LIN {X 0,Y 176.347,Z 623.439,A -85,B 0,C 180,E1 -22419.173,E2 -22419.173} C_VEL
LIN {X 0,Y 177.506,Z 621.11,A -85,B 0,C 180,E1 -22423.742,E2 -22423.742} C_VEL
LIN {X 0,Y 179.733,Z 617.398,A -85,B 0,C 180,E1 -22428.229,E2 -22428.229} C_VEL
LIN {X 0,Y 182.863,Z 612.047,A -85,B 0,C 180,E1 -22432.722,E2 -22432.722} C_VEL
LIN {X 0,Y 186.944,Z 605.294,A -85,B 0,C 180,E1 -22436.815,E2 -22436.815} C_VEL
LIN {X 0,Y 191.406,Z 597.669,A -85,B 0,C 180,E1 -22440.322,E2 -22440.322} C_VEL
LIN {X 0,Y 195.831,Z 589.742,A -85,B 0,C 180,E1 -22443.18,E2 -22443.18} C_VEL
LIN {X 0,Y 200.702,Z 580.202,A -85,B 0,C 180,E1 -22445.911,E2 -22445.911} C_VEL
LIN {X 0,Y 205.489,Z 569.651,A -85,B 0,C 180,E1 -22448.308,E2 -22448.308} C_VEL
LIN {X 0,Y 210.252,Z 558.007,A -85,B 0,C 180,E1 -22450.363,E2 -22450.363} C_VEL
LIN {X 0,Y 214.231,Z 546.657,A -85,B 0,C 180,E1 -22451.943,E2 -22451.943} C_VEL
LIN {X 0,Y 217.948,Z 534.375,A -85,B 0,C 180,E1 -22453.252,E2 -22453.252} C_VEL
LIN {X 0,Y 221.215,Z 520.802,A -85,B 0,C 180,E1 -22454.34,E2 -22454.34} C_VEL
LIN {X 0,Y 223.705,Z 506.759,A -85,B 0,C 180,E1 -22455.138,E2 -22455.138} C_VEL
LIN {X 0,Y 225.13,Z 493.571,A -85,B 0,C 180,E1 -22455.648,E2 -22455.648} C_VEL
LIN {X 0,Y 228.62,Z 440.792,A -85,B 0,C 180,E1 -22457.146,E2 -22457.146} C_VEL
LIN {X 0,Y 223.879,Z 429.35,A -85,B 0,C 180,E1 -22459.176,E2 -22459.176} C_VEL
LIN {X 0,Y 218.405,Z 417.952,A -85,B 0,C 180,E1 -22461.66,E2 -22461.66} C_VEL
LIN {X 0,Y 213.133,Z 408.172,A -85,B 0,C 180,E1 -22464.263,E2 -22464.263} C_VEL
LIN {X 0,Y 208.258,Z 399.763,A -85,B 0,C 180,E1 -22466.934,E2 -22466.934} C_VEL
LIN {X 0,Y 204.902,Z 394.49,A -85,B 0,C 180,E1 -22468.95,E2 -22468.95} C_VEL
LIN {X 0,Y 201.919,Z 389.944,A -85,B 0,C 180,E1 -22470.91,E2 -22470.91} C_VEL
LIN {X 0,Y 198.244,Z 384.689,A -85,B 0,C 180,E1 -22473.59,E2 -22473.59} C_VEL
LIN {X 0,Y 195.498,Z 381.922,A -85,B 0,C 180,E1 -22475.76,E2 -22475.76} C_VEL
LIN {X 0,Y 194.093,Z 379.464,A -85,B 0,C 180,E1 -22477.093,E2 -22477.093} C_VEL
LIN {X 0,Y 191.265,Z 377.162,A -85,B 0,C 180,E1 -22479.815,E2 -22479.815} C_VEL
LIN {X 0,Y 189.615,Z 374.053,A -85,B 0,C 180,E1 -22481.903,E2 -22481.903} C_VEL
LIN {X 0,Y 186.176,Z 371.524,A -85,B 0,C 180,E1 -22486.91,E2 -22486.91} C_VEL
LIN {X 0,Y 185.017,Z 368.902,A -85,B 0,C 180,E1 -22489.847,E2 -22489.847} C_VEL
LIN {X 0,Y 184.851,Z 367.99,A -85,B 0,C 180,E1 -22490.546,E2 -22490.546} C_VEL
LIN {X 0,Y 183.865,Z 367.537,A -85,B 0,C 180,E1 -22500.001,E2 -22500.001} C_VEL
LIN {X 0,Y 184.86,Z 368.103,A -85,B 0,C 180,E1 -22503.952,E2 -22503.952} C_VEL
LIN {X 0,Y 186.113,Z 371.068,A -85,B 0,C 180,E1 -22507.323,E2 -22507.323} C_VEL
LIN {X 0,Y 188.809,Z 373.526,A -85,B 0,C 180,E1 -22511.542,E2 -22511.542} C_VEL
LIN {X 0,Y 189.74,Z 374.056,A -85,B 0,C 180,E1 -22512.671,E2 -22512.671} C_VEL
LIN {X 0,Y 191.233,Z 376.977,A -85,B 0,C 180,E1 -22514.568,E2 -22514.568} C_VEL
LIN {X 0,Y 194.282,Z 379.772,A -85,B 0,C 180,E1 -22517.526,E2 -22517.526} C_VEL
LIN {X 0,Y 196.429,Z 383.09,A -85,B 0,C 180,E1 -22519.463,E2 -22519.463} C_VEL
LIN {X 0,Y 198.609,Z 385.225,A -85,B 0,C 180,E1 -22521.131,E2 -22521.131} C_VEL
LIN {X 0,Y 201.298,Z 388.85,A -85,B 0,C 180,E1 -22523.083,E2 -22523.083} C_VEL
LIN {X 0,Y 202.611,Z 390.385,A -85,B 0,C 180,E1 -22523.951,E2 -22523.951} C_VEL
LIN {X 0,Y 206.418,Z 395.562,A -85,B 0,C 180,E1 -22526.329,E2 -22526.329} C_VEL
LIN {X 0,Y 210.161,Z 400.809,A -85,B 0,C 180,E1 -22528.441,E2 -22528.441} C_VEL
LIN {X 0,Y 214.285,Z 406.702,A -85,B 0,C 180,E1 -22530.555,E2 -22530.555} C_VEL
LIN {X 0,Y 221.11,Z 417.678,A -85,B 0,C 180,E1 -22533.724,E2 -22533.724} C_VEL
LIN {X 0,Y 224.783,Z 424.595,A -85,B 0,C 180,E1 -22535.312,E2 -22535.312} C_VEL
LIN {X 0,Y 229.084,Z 433.995,A -85,B 0,C 180,E1 -22537.104,E2 -22537.104} C_VEL
LIN {X 0,Y 225.117,Z 490.442,A -85,B 0,C 180,E1 -22538.697,E2 -22538.697} C_VEL
LIN {X 0,Y 223.295,Z 504.424,A -85,B 0,C 180,E1 -22539.378,E2 -22539.378} C_VEL
LIN {X 0,Y 220.715,Z 518.004,A -85,B 0,C 180,E1 -22540.342,E2 -22540.342} C_VEL
LIN {X 0,Y 217.324,Z 531.263,A -85,B 0,C 180,E1 -22541.599,E2 -22541.599} C_VEL
LIN {X 0,Y 213.305,Z 544.035,A -85,B 0,C 180,E1 -22543.201,E2 -22543.201} C_VEL
LIN {X 0,Y 208.902,Z 555.625,A -85,B 0,C 180,E1 -22545.051,E2 -22545.051} C_VEL
LIN {X 0,Y 204.242,Z 566.232,A -85,B 0,C 180,E1 -22547.189,E2 -22547.189} C_VEL
LIN {X 0,Y 199.25,Z 576.745,A -85,B 0,C 180,E1 -22549.932,E2 -22549.932} C_VEL
LIN {X 0,Y 194.962,Z 584.9,A -85,B 0,C 180,E1 -22552.627,E2 -22552.627} C_VEL
LIN {X 0,Y 190.644,Z 592.537,A -85,B 0,C 180,E1 -22555.794,E2 -22555.794} C_VEL
LIN {X 0,Y 186.448,Z 599.361,A -85,B 0,C 180,E1 -22559.412,E2 -22559.412} C_VEL
LIN {X 0,Y 182.571,Z 605.398,A -85,B 0,C 180,E1 -22563.725,E2 -22563.725} C_VEL
LIN {X 0,Y 180.255,Z 608.851,A -85,B 0,C 180,E1 -22567.053,E2 -22567.053} C_VEL
LIN {X 0,Y 178.042,Z 612.15,A -85,B 0,C 180,E1 -22571.592,E2 -22571.592} C_VEL
LIN {X 0,Y 176.557,Z 614.028,A -85,B 0,C 180,E1 -22576.183,E2 -22576.183} C_VEL
LIN {X 0,Y 175.955,Z 614.552,A -85,B 0,C 180,E1 -22580.807,E2 -22580.807} C_VEL
LIN {X 0,Y 176.019,Z 613.752,A -85,B 0,C 180,E1 -22585.42,E2 -22585.42} C_VEL
LIN {X 0,Y 176.277,Z 611.638,A -85,B 0,C 180,E1 -22590,E2 -22590} C_VEL
LIN {X 0,Y 177.061,Z 608.156,A -85,B 0,C 180,E1 -22594.553,E2 -22594.553} C_VEL
LIN {X 0,Y 178.635,Z 603.197,A -85,B 0,C 180,E1 -22599.054,E2 -22599.054} C_VEL
LIN {X 0,Y 180.415,Z 598.399,A -85,B 0,C 180,E1 -22602.371,E2 -22602.371} C_VEL
LIN {X 0,Y 182.925,Z 591.954,A -85,B 0,C 180,E1 -22605.931,E2 -22605.931} C_VEL
LIN {X 0,Y 185.824,Z 584.276,A -85,B 0,C 180,E1 -22609.325,E2 -22609.325} C_VEL
LIN {X 0,Y 189.093,Z 575.604,A -85,B 0,C 180,E1 -22612.392,E2 -22612.392} C_VEL
LIN {X 0,Y 192.844,Z 565.1,A -85,B 0,C 180,E1 -22615.354,E2 -22615.354} C_VEL
LIN {X 0,Y 196.711,Z 553.334,A -85,B 0,C 180,E1 -22617.964,E2 -22617.964} C_VEL
LIN {X 0,Y 200.089,Z 541.52,A -85,B 0,C 180,E1 -22620.034,E2 -22620.034} C_VEL
LIN {X 0,Y 202.809,Z 530.234,A -85,B 0,C 180,E1 -22621.609,E2 -22621.609} C_VEL
LIN {X 0,Y 205.621,Z 517.023,A -85,B 0,C 180,E1 -22623.005,E2 -22623.005} C_VEL
LIN {X 0,Y 207.715,Z 503.456,A -85,B 0,C 180,E1 -22624.082,E2 -22624.082} C_VEL
LIN {X 0,Y 209.146,Z 489.592,A -85,B 0,C 180,E1 -22624.837,E2 -22624.837} C_VEL
LIN {X 0,Y 213.093,Z 419.656,A -85,B 0,C 180,E1 -22627.034,E2 -22627.034} C_VEL
LIN {X 0,Y 208.609,Z 408.771,A -85,B 0,C 180,E1 -22628.586,E2 -22628.586} C_VEL
LIN {X 0,Y 200.689,Z 394.452,A -85,B 0,C 180,E1 -22631.361,E2 -22631.361} C_VEL
LIN {X 0,Y 193.602,Z 383.533,A -85,B 0,C 180,E1 -22634.066,E2 -22634.066} C_VEL
LIN {X 0,Y 188.109,Z 375.762,A -85,B 0,C 180,E1 -22636.369,E2 -22636.369} C_VEL
LIN {X 0,Y 185.242,Z 371.796,A -85,B 0,C 180,E1 -22637.667,E2 -22637.667} C_VEL
LIN {X 0,Y 182.829,Z 368.831,A -85,B 0,C 180,E1 -22638.797,E2 -22638.797} C_VEL
LIN {X 0,Y 181.921,Z 367.135,A -85,B 0,C 180,E1 -22639.275,E2 -22639.275} C_VEL
LIN {X 0,Y 179.566,Z 364.991,A -85,B 0,C 180,E1 -22640.413,E2 -22640.413} C_VEL
LIN {X 0,Y 178.526,Z 362.549,A -85,B 0,C 180,E1 -22641.036,E2 -22641.036} C_VEL
LIN {X 0,Y 178.411,Z 361.88,A -85,B 0,C 180,E1 -22641.24,E2 -22641.24} C_VEL
LIN {X 0,Y 178.483,Z 361.865,A -85,B 0,C 180,E1 -22646.545,E2 -22646.545} C_VEL
LIN {X 0,Y 178.519,Z 361.868,A -85,B 0,C 180,E1 -22650.006,E2 -22650.006} C_VEL
LIN {X 0,Y 178.517,Z 361.866,A -85,B 0,C 180,E1 -22654.885,E2 -22654.885} C_VEL
LIN {X 0,Y 178.603,Z 361.846,A -85,B 0,C 180,E1 -22661.65,E2 -22661.65} C_VEL
LIN {X 0,Y 178.633,Z 361.829,A -85,B 0,C 180,E1 -22666.345,E2 -22666.345} C_VEL
LIN {X 0,Y 178.901,Z 361.824,A -85,B 0,C 180,E1 -22670.958,E2 -22670.958} C_VEL
LIN {X 0,Y 179.119,Z 361.78,A -85,B 0,C 180,E1 -22677.751,E2 -22677.751} C_VEL
LIN {X 0,Y 179.332,Z 361.773,A -85,B 0,C 180,E1 -22679.999,E2 -22679.999} C_VEL
LIN {X 0,Y 178.884,Z 361.827,A -85,B 0,C 180,E1 -22686.768,E2 -22686.768} C_VEL
LIN {X 0,Y 178.827,Z 361.819,A -85,B 0,C 180,E1 -22690.74,E2 -22690.74} C_VEL
LIN {X 0,Y 178.585,Z 361.846,A -85,B 0,C 180,E1 -22695.99,E2 -22695.99} C_VEL
LIN {X 0,Y 178.552,Z 361.864,A -85,B 0,C 180,E1 -22699.154,E2 -22699.154} C_VEL
LIN {X 0,Y 178.51,Z 361.862,A -85,B 0,C 180,E1 -22705.111,E2 -22705.111} C_VEL
LIN {X 0,Y 178.455,Z 361.87,A -85,B 0,C 180,E1 -22710.795,E2 -22710.795} C_VEL
LIN {X 0,Y 178.47,Z 361.887,A -85,B 0,C 180,E1 -22712.531,E2 -22712.531} C_VEL
LIN {X 0,Y 179.25,Z 364.296,A -85,B 0,C 180,E1 -22713.04,E2 -22713.04} C_VEL
LIN {X 0,Y 181.077,Z 366.543,A -85,B 0,C 180,E1 -22713.972,E2 -22713.972} C_VEL
LIN {X 0,Y 182.337,Z 367.607,A -85,B 0,C 180,E1 -22714.562,E2 -22714.562} C_VEL
LIN {X 0,Y 184.25,Z 370.718,A -85,B 0,C 180,E1 -22715.52,E2 -22715.52} C_VEL
LIN {X 0,Y 185.968,Z 372.684,A -85,B 0,C 180,E1 -22716.297,E2 -22716.297} C_VEL
LIN {X 0,Y 188.777,Z 376.476,A -85,B 0,C 180,E1 -22717.546,E2 -22717.546} C_VEL
LIN {X 0,Y 194.692,Z 386.533,A -85,B 0,C 180,E1 -22720.08,E2 -22720.08} C_VEL
LIN {X 0,Y 201.001,Z 398.408,A -85,B 0,C 180,E1 -22722.559,E2 -22722.559} C_VEL
LIN {X 0,Y 206.826,Z 411.246,A -85,B 0,C 180,E1 -22724.717,E2 -22724.717} C_VEL
LIN {X 0,Y 212.704,Z 426.479,A -85,B 0,C 180,E1 -22726.81,E2 -22726.81} C_VEL
LIN {X 0,Y 212.485,Z 434.308,A -85,B 0,C 180,E1 -22727.099,E2 -22727.099} C_VEL
LIN {X 0,Y 210.836,Z 461.914,A -85,B 0,C 180,E1 -22727.922,E2 -22727.922} C_VEL
LIN {X 0,Y 209.983,Z 467.763,A -85,B 0,C 180,E1 -22727.981,E2 -22727.981} C_VEL
LIN {X 0,Y 204.53,Z 486.79,A -85,B 0,C 180,E1 -22727.57,E2 -22727.57} C_VEL
LIN {X 0,Y 203.628,Z 492.629,A -85,B 0,C 180,E1 -22727.646,E2 -22727.646} C_VEL
LIN {X 0,Y 202.346,Z 506.62,A -85,B 0,C 180,E1 -22728.254,E2 -22728.254} C_VEL
LIN {X 0,Y 200.244,Z 520.531,A -85,B 0,C 180,E1 -22729.181,E2 -22729.181} C_VEL
LIN {X 0,Y 197.387,Z 534.321,A -85,B 0,C 180,E1 -22730.474,E2 -22730.474} C_VEL
LIN {X 0,Y 194.258,Z 546.758,A -85,B 0,C 180,E1 -22732.047,E2 -22732.047} C_VEL
LIN {X 0,Y 190.491,Z 559.651,A -85,B 0,C 180,E1 -22734.176,E2 -22734.176} C_VEL
LIN {X 0,Y 186.997,Z 569.993,A -85,B 0,C 180,E1 -22736.335,E2 -22736.335} C_VEL
LIN {X 0,Y 183.467,Z 579.723,A -85,B 0,C 180,E1 -22738.86,E2 -22738.86} C_VEL
LIN {X 0,Y 179.689,Z 589.461,A -85,B 0,C 180,E1 -22742.009,E2 -22742.009} C_VEL
LIN {X 0,Y 176.498,Z 597.532,A -85,B 0,C 180,E1 -22745.286,E2 -22745.286} C_VEL
LIN {X 0,Y 173.566,Z 605.272,A -85,B 0,C 180,E1 -22749.25,E2 -22749.25} C_VEL
LIN {X 0,Y 171.381,Z 611.465,A -85,B 0,C 180,E1 -22753.319,E2 -22753.319} C_VEL
LIN {X 0,Y 170.039,Z 615.675,A -85,B 0,C 180,E1 -22756.861,E2 -22756.861} C_VEL
LIN {X 0,Y 169.291,Z 619.025,A -85,B 0,C 180,E1 -22760.442,E2 -22760.442} C_VEL
LIN {X 0,Y 168.872,Z 622.15,A -85,B 0,C 180,E1 -22765.226,E2 -22765.226} C_VEL
LIN {X 0,Y 168.885,Z 623.187,A -85,B 0,C 180,E1 -22767.615,E2 -22767.615} C_VEL
LIN {X 0,Y 168.999,Z 623.881,A -85,B 0,C 180,E1 -22770,E2 -22770} C_VEL
LIN {X 0,Y 168.857,Z 624.241,A -85,B 0,C 180,E1 -22774.775,E2 -22774.775} C_VEL
LIN {X 0,Y 169.315,Z 623.275,A -85,B 0,C 180,E1 -22779.557,E2 -22779.557} C_VEL
LIN {X 0,Y 170.568,Z 620.977,A -85,B 0,C 180,E1 -22784.313,E2 -22784.313} C_VEL
LIN {X 0,Y 172.941,Z 617.296,A -85,B 0,C 180,E1 -22788.971,E2 -22788.971} C_VEL
LIN {X 0,Y 176.187,Z 612.126,A -85,B 0,C 180,E1 -22793.508,E2 -22793.508} C_VEL
LIN {X 0,Y 179.414,Z 607.14,A -85,B 0,C 180,E1 -22796.774,E2 -22796.774} C_VEL
LIN {X 0,Y 183.861,Z 600.02,A -85,B 0,C 180,E1 -22800.428,E2 -22800.428} C_VEL
LIN {X 0,Y 188.274,Z 592.588,A -85,B 0,C 180,E1 -22803.407,E2 -22803.407} C_VEL
LIN {X 0,Y 193.292,Z 583.68,A -85,B 0,C 180,E1 -22806.216,E2 -22806.216} C_VEL
LIN {X 0,Y 198.071,Z 573.961,A -85,B 0,C 180,E1 -22808.684,E2 -22808.684} C_VEL
LIN {X 0,Y 202.892,Z 563.197,A -85,B 0,C 180,E1 -22810.828,E2 -22810.828} C_VEL
LIN {X 0,Y 207.421,Z 551.539,A -85,B 0,C 180,E1 -22812.659,E2 -22812.659} C_VEL
LIN {X 0,Y 211.743,Z 538.704,A -85,B 0,C 180,E1 -22814.186,E2 -22814.186} C_VEL
LIN {X 0,Y 215.364,Z 525.362,A -85,B 0,C 180,E1 -22815.381,E2 -22815.381} C_VEL
LIN {X 0,Y 218.181,Z 511.58,A -85,B 0,C 180,E1 -22816.28,E2 -22816.28} C_VEL
LIN {X 0,Y 220.114,Z 497.18,A -85,B 0,C 180,E1 -22816.916,E2 -22816.916} C_VEL
LIN {X 0,Y 223.975,Z 443.363,A -85,B 0,C 180,E1 -22818.439,E2 -22818.439} C_VEL
LIN {X 0,Y 219.593,Z 432.728,A -85,B 0,C 180,E1 -22820.437,E2 -22820.437} C_VEL
LIN {X 0,Y 214.834,Z 422.604,A -85,B 0,C 180,E1 -22822.734,E2 -22822.734} C_VEL
LIN {X 0,Y 209.923,Z 413.205,A -85,B 0,C 180,E1 -22825.31,E2 -22825.31} C_VEL
LIN {X 0,Y 204.972,Z 404.476,A -85,B 0,C 180,E1 -22828.202,E2 -22828.202} C_VEL
LIN {X 0,Y 202.27,Z 400.161,A -85,B 0,C 180,E1 -22829.928,E2 -22829.928} C_VEL
LIN {X 0,Y 199.369,Z 395.626,A -85,B 0,C 180,E1 -22831.951,E2 -22831.951} C_VEL
LIN {X 0,Y 196.225,Z 391.115,A -85,B 0,C 180,E1 -22834.369,E2 -22834.369} C_VEL
LIN {X 0,Y 193.505,Z 388.049,A -85,B 0,C 180,E1 -22836.665,E2 -22836.665} C_VEL
LIN {X 0,Y 192.296,Z 386.084,A -85,B 0,C 180,E1 -22837.859,E2 -22837.859} C_VEL
LIN {X 0,Y 189.57,Z 383.514,A -85,B 0,C 180,E1 -22840.676,E2 -22840.676} C_VEL
LIN {X 0,Y 188.133,Z 380.752,A -85,B 0,C 180,E1 -22842.612,E2 -22842.612} C_VEL
LIN {X 0,Y 185.178,Z 378.541,A -85,B 0,C 180,E1 -22847.117,E2 -22847.117} C_VEL
LIN {X 0,Y 183.971,Z 375.813,A -85,B 0,C 180,E1 -22850.314,E2 -22850.314} C_VEL
LIN {X 0,Y 183.753,Z 374.963,A -85,B 0,C 180,E1 -22851.201,E2 -22851.201} C_VEL
LIN {X 0,Y 182.999,Z 374.568,A -85,B 0,C 180,E1 -22860.001,E2 -22860.001} C_VEL
LIN {X 0,Y 183.852,Z 375.08,A -85,B 0,C 180,E1 -22863.562,E2 -22863.562} C_VEL
LIN {X 0,Y 185.105,Z 378.074,A -85,B 0,C 180,E1 -22867.089,E2 -22867.089} C_VEL
LIN {X 0,Y 187.956,Z 380.602,A -85,B 0,C 180,E1 -22871.595,E2 -22871.595} C_VEL
LIN {X 0,Y 188.5,Z 381.338,A -85,B 0,C 180,E1 -22872.329,E2 -22872.329} C_VEL
LIN {X 0,Y 190.352,Z 384.369,A -85,B 0,C 180,E1 -22874.637,E2 -22874.637} C_VEL
LIN {X 0,Y 192.699,Z 386.55,A -85,B 0,C 180,E1 -22876.965,E2 -22876.965} C_VEL
LIN {X 0,Y 194.824,Z 389.778,A -85,B 0,C 180,E1 -22878.946,E2 -22878.946} C_VEL
LIN {X 0,Y 196.77,Z 391.782,A -85,B 0,C 180,E1 -22880.5,E2 -22880.5} C_VEL
LIN {X 0,Y 199.598,Z 395.55,A -85,B 0,C 180,E1 -22882.618,E2 -22882.618} C_VEL
LIN {X 0,Y 204.059,Z 401.66,A -85,B 0,C 180,E1 -22885.569,E2 -22885.569} C_VEL
LIN {X 0,Y 209.178,Z 409.019,A -85,B 0,C 180,E1 -22888.531,E2 -22888.531} C_VEL
LIN {X 0,Y 214.446,Z 417.321,A -85,B 0,C 180,E1 -22891.245,E2 -22891.245} C_VEL
LIN {X 0,Y 219.675,Z 426.375,A -85,B 0,C 180,E1 -22893.689,E2 -22893.689} C_VEL
LIN {X 0,Y 224.384,Z 436.682,A -85,B 0,C 180,E1 -22895.793,E2 -22895.793} C_VEL
LIN {X 0,Y 220.468,Z 490.541,A -85,B 0,C 180,E1 -22897.325,E2 -22897.325} C_VEL
LIN {X 0,Y 218.601,Z 504.443,A -85,B 0,C 180,E1 -22898.001,E2 -22898.001} C_VEL
LIN {X 0,Y 215.865,Z 518.316,A -85,B 0,C 180,E1 -22898.987,E2 -22898.987} C_VEL
LIN {X 0,Y 212.103,Z 532.442,A -85,B 0,C 180,E1 -22900.352,E2 -22900.352} C_VEL
LIN {X 0,Y 207.937,Z 545.022,A -85,B 0,C 180,E1 -22901.965,E2 -22901.965} C_VEL
LIN {X 0,Y 203.366,Z 556.527,A -85,B 0,C 180,E1 -22903.847,E2 -22903.847} C_VEL
LIN {X 0,Y 198.103,Z 567.943,A -85,B 0,C 180,E1 -22906.23,E2 -22906.23} C_VEL
LIN {X 0,Y 192.935,Z 578.139,A -85,B 0,C 180,E1 -22909.03,E2 -22909.03} C_VEL
LIN {X 0,Y 188.108,Z 586.801,A -85,B 0,C 180,E1 -22912.068,E2 -22912.068} C_VEL
LIN {X 0,Y 183.371,Z 594.596,A -85,B 0,C 180,E1 -22915.577,E2 -22915.577} C_VEL
LIN {X 0,Y 179.128,Z 601.026,A -85,B 0,C 180,E1 -22919.334,E2 -22919.334} C_VEL
LIN {X 0,Y 175.196,Z 606.7,A -85,B 0,C 180,E1 -22923.816,E2 -22923.816} C_VEL
LIN {X 0,Y 172.28,Z 610.785,A -85,B 0,C 180,E1 -22928.461,E2 -22928.461} C_VEL
LIN {X 0,Y 170.278,Z 613.41,A -85,B 0,C 180,E1 -22933.207,E2 -22933.207} C_VEL
LIN {X 0,Y 169.121,Z 614.65,A -85,B 0,C 180,E1 -22938.008,E2 -22938.008} C_VEL
LIN {X 0,Y 168.831,Z 614.547,A -85,B 0,C 180,E1 -22942.826,E2 -22942.826} C_VEL
LIN {X 0,Y 168.983,Z 613.555,A -85,B 0,C 180,E1 -22946.543,E2 -22946.543} C_VEL
LIN {X 0,Y 169.177,Z 611.922,A -85,B 0,C 180,E1 -22950,E2 -22950} C_VEL
LIN {X 0,Y 170.002,Z 608.478,A -85,B 0,C 180,E1 -22954.743,E2 -22954.743} C_VEL
LIN {X 0,Y 171.648,Z 603.56,A -85,B 0,C 180,E1 -22959.426,E2 -22959.426} C_VEL
LIN {X 0,Y 173.514,Z 598.806,A -85,B 0,C 180,E1 -22962.871,E2 -22962.871} C_VEL
LIN {X 0,Y 176.126,Z 592.409,A -85,B 0,C 180,E1 -22966.563,E2 -22966.563} C_VEL
LIN {X 0,Y 179.164,Z 584.785,A -85,B 0,C 180,E1 -22970.073,E2 -22970.073} C_VEL
LIN {X 0,Y 182.581,Z 576.175,A -85,B 0,C 180,E1 -22973.237,E2 -22973.237} C_VEL
LIN {X 0,Y 186.482,Z 565.745,A -85,B 0,C 180,E1 -22976.283,E2 -22976.283} C_VEL
LIN {X 0,Y 190.512,Z 554.068,A -85,B 0,C 180,E1 -22978.958,E2 -22978.958} C_VEL
LIN {X 0,Y 194.008,Z 542.371,A -85,B 0,C 180,E1 -22981.077,E2 -22981.077} C_VEL
LIN {X 0,Y 196.833,Z 531.239,A -85,B 0,C 180,E1 -22982.686,E2 -22982.686} C_VEL
LIN {X 0,Y 199.719,Z 518.257,A -85,B 0,C 180,E1 -22984.112,E2 -22984.112} C_VEL
LIN {X 0,Y 202.031,Z 504.288,A -85,B 0,C 180,E1 -22985.256,E2 -22985.256} C_VEL
LIN {X 0,Y 203.634,Z 489.716,A -85,B 0,C 180,E1 -22986.068,E2 -22986.068} C_VEL
LIN {X 0,Y 207.648,Z 421.746,A -85,B 0,C 180,E1 -22988.234,E2 -22988.234} C_VEL
LIN {X 0,Y 203.963,Z 412.813,A -85,B 0,C 180,E1 -22989.582,E2 -22989.582} C_VEL
LIN {X 0,Y 196.447,Z 399.021,A -85,B 0,C 180,E1 -22992.367,E2 -22992.367} C_VEL
LIN {X 0,Y 189.899,Z 388.695,A -85,B 0,C 180,E1 -22995.008,E2 -22995.008} C_VEL
LIN {X 0,Y 184.401,Z 380.876,A -85,B 0,C 180,E1 -22997.439,E2 -22997.439} C_VEL
LIN {X 0,Y 181.917,Z 377.414,A -85,B 0,C 180,E1 -22998.626,E2 -22998.626} C_VEL
LIN {X 0,Y 179.282,Z 373.775,A -85,B 0,C 180,E1 -22999.955,E2 -22999.955} C_VEL
LIN {X 0,Y 176.045,Z 369.846,A -85,B 0,C 180,E1 -23001.668,E2 -23001.668} C_VEL
LIN {X 0,Y 175.131,Z 368.165,A -85,B 0,C 180,E1 -23002.217,E2 -23002.217} C_VEL
LIN {X 0,Y 172.807,Z 366.225,A -85,B 0,C 180,E1 -23003.501,E2 -23003.501} C_VEL
LIN {X 0,Y 171.609,Z 363.889,A -85,B 0,C 180,E1 -23004.296,E2 -23004.296} C_VEL
LIN {X 0,Y 171.402,Z 362.761,A -85,B 0,C 180,E1 -23004.517,E2 -23004.517} C_VEL
LIN {X 0,Y 171.454,Z 362.753,A -85,B 0,C 180,E1 -23009.404,E2 -23009.404} C_VEL
LIN {X 0,Y 171.455,Z 362.738,A -85,B 0,C 180,E1 -23014.39,E2 -23014.39} C_VEL
LIN {X 0,Y 171.503,Z 362.721,A -85,B 0,C 180,E1 -23020.862,E2 -23020.862} C_VEL
LIN {X 0,Y 171.548,Z 362.716,A -85,B 0,C 180,E1 -23025.769,E2 -23025.769} C_VEL
LIN {X 0,Y 171.84,Z 362.701,A -85,B 0,C 180,E1 -23030.584,E2 -23030.584} C_VEL
LIN {X 0,Y 171.78,Z 362.677,A -85,B 0,C 180,E1 -23035.306,E2 -23035.306} C_VEL
LIN {X 0,Y 172.297,Z 362.649,A -85,B 0,C 180,E1 -23039.999,E2 -23039.999} C_VEL
LIN {X 0,Y 171.848,Z 362.702,A -85,B 0,C 180,E1 -23047.047,E2 -23047.047} C_VEL
LIN {X 0,Y 171.762,Z 362.7,A -85,B 0,C 180,E1 -23050.893,E2 -23050.893} C_VEL
LIN {X 0,Y 171.515,Z 362.729,A -85,B 0,C 180,E1 -23056.668,E2 -23056.668} C_VEL
LIN {X 0,Y 171.426,Z 362.738,A -85,B 0,C 180,E1 -23061.652,E2 -23061.652} C_VEL
LIN {X 0,Y 171.438,Z 362.74,A -85,B 0,C 180,E1 -23065.598,E2 -23065.598} C_VEL
LIN {X 0,Y 171.393,Z 362.754,A -85,B 0,C 180,E1 -23069.139,E2 -23069.139} C_VEL
LIN {X 0,Y 172.218,Z 365.23,A -85,B 0,C 180,E1 -23069.761,E2 -23069.761} C_VEL
LIN {X 0,Y 174.231,Z 367.566,A -85,B 0,C 180,E1 -23070.945,E2 -23070.945} C_VEL
LIN {X 0,Y 175.498,Z 368.552,A -85,B 0,C 180,E1 -23071.624,E2 -23071.624} C_VEL
LIN {X 0,Y 177.334,Z 371.605,A -85,B 0,C 180,E1 -23072.681,E2 -23072.681} C_VEL
LIN {X 0,Y 179.414,Z 373.847,A -85,B 0,C 180,E1 -23073.743,E2 -23073.743} C_VEL
LIN {X 0,Y 181.908,Z 377.31,A -85,B 0,C 180,E1 -23075,E2 -23075} C_VEL
LIN {X 0,Y 186.177,Z 383.317,A -85,B 0,C 180,E1 -23077.006,E2 -23077.006} C_VEL
LIN {X 0,Y 192.863,Z 395.199,A -85,B 0,C 180,E1 -23079.961,E2 -23079.961} C_VEL
LIN {X 0,Y 198.523,Z 406.729,A -85,B 0,C 180,E1 -23082.269,E2 -23082.269} C_VEL
LIN {X 0,Y 203.237,Z 417.815,A -85,B 0,C 180,E1 -23084.101,E2 -23084.101} C_VEL
LIN {X 0,Y 207.328,Z 428.823,A -85,B 0,C 180,E1 -23085.645,E2 -23085.645} C_VEL
LIN {X 0,Y 203.628,Z 492.629,A -85,B 0,C 180,E1 -23087.646,E2 -23087.646} C_VEL
LIN {X 0,Y 202.628,Z 498.447,A -85,B 0,C 180,E1 -23087.725,E2 -23087.725} C_VEL
LIN {X 0,Y 199.3,Z 507.809,A -85,B 0,C 180,E1 -23087.657,E2 -23087.657} C_VEL
LIN {X 0,Y 195.715,Z 517.089,A -85,B 0,C 180,E1 -23087.74,E2 -23087.74} C_VEL
LIN {X 0,Y 194.266,Z 522.644,A -85,B 0,C 180,E1 -23088.083,E2 -23088.083} C_VEL
LIN {X 0,Y 191.478,Z 535.361,A -85,B 0,C 180,E1 -23089.347,E2 -23089.347} C_VEL
LIN {X 0,Y 188.218,Z 547.542,A -85,B 0,C 180,E1 -23090.943,E2 -23090.943} C_VEL
LIN {X 0,Y 184.701,Z 559.07,A -85,B 0,C 180,E1 -23092.899,E2 -23092.899} C_VEL
LIN {X 0,Y 181.116,Z 569.383,A -85,B 0,C 180,E1 -23095.086,E2 -23095.086} C_VEL
LIN {X 0,Y 177.372,Z 579.178,A -85,B 0,C 180,E1 -23097.663,E2 -23097.663} C_VEL
LIN {X 0,Y 173.393,Z 588.972,A -85,B 0,C 180,E1 -23100.898,E2 -23100.898} C_VEL
LIN {X 0,Y 170.034,Z 597.094,A -85,B 0,C 180,E1 -23104.279,E2 -23104.279} C_VEL
LIN {X 0,Y 166.875,Z 604.874,A -85,B 0,C 180,E1 -23108.377,E2 -23108.377} C_VEL
LIN {X 0,Y 164.544,Z 611.108,A -85,B 0,C 180,E1 -23112.604,E2 -23112.604} C_VEL
LIN {X 0,Y 162.739,Z 616.602,A -85,B 0,C 180,E1 -23117.53,E2 -23117.53} C_VEL
LIN {X 0,Y 161.926,Z 620.494,A -85,B 0,C 180,E1 -23122.519,E2 -23122.519} C_VEL
LIN {X 0,Y 161.795,Z 622.947,A -85,B 0,C 180,E1 -23127.511,E2 -23127.511} C_VEL
LIN {X 0,Y 161.91,Z 623.657,A -85,B 0,C 180,E1 -23130,E2 -23130} C_VEL
LIN {X 0,Y 161.795,Z 624.019,A -85,B 0,C 180,E1 -23132.49,E2 -23132.49} C_VEL
LIN {X 0,Y 161.927,Z 623.743,A -85,B 0,C 180,E1 -23137.481,E2 -23137.481} C_VEL
LIN {X 0,Y 162.85,Z 622.145,A -85,B 0,C 180,E1 -23142.461,E2 -23142.461} C_VEL
LIN {X 0,Y 164.832,Z 619.198,A -85,B 0,C 180,E1 -23147.365,E2 -23147.365} C_VEL
LIN {X 0,Y 167.854,Z 614.821,A -85,B 0,C 180,E1 -23152.137,E2 -23152.137} C_VEL
LIN {X 0,Y 170.735,Z 610.512,A -85,B 0,C 180,E1 -23155.607,E2 -23155.607} C_VEL
LIN {X 0,Y 174.996,Z 604.265,A -85,B 0,C 180,E1 -23159.469,E2 -23159.469} C_VEL
LIN {X 0,Y 179.965,Z 596.505,A -85,B 0,C 180,E1 -23163.142,E2 -23163.142} C_VEL
LIN {X 0,Y 184.938,Z 588.423,A -85,B 0,C 180,E1 -23166.087,E2 -23166.087} C_VEL
LIN {X 0,Y 190.344,Z 578.703,A -85,B 0,C 180,E1 -23168.878,E2 -23168.878} C_VEL
LIN {X 0,Y 195.534,Z 567.938,A -85,B 0,C 180,E1 -23171.332,E2 -23171.332} C_VEL
LIN {X 0,Y 200.657,Z 556.027,A -85,B 0,C 180,E1 -23173.42,E2 -23173.42} C_VEL
LIN {X 0,Y 205.039,Z 544.319,A -85,B 0,C 180,E1 -23174.986,E2 -23174.986} C_VEL
LIN {X 0,Y 209.298,Z 530.526,A -85,B 0,C 180,E1 -23176.388,E2 -23176.388} C_VEL
LIN {X 0,Y 212.62,Z 516.364,A -85,B 0,C 180,E1 -23177.432,E2 -23177.432} C_VEL
LIN {X 0,Y 214.805,Z 503.498,A -85,B 0,C 180,E1 -23178.1,E2 -23178.1} C_VEL
LIN {X 0,Y 216.417,Z 487.474,A -85,B 0,C 180,E1 -23178.628,E2 -23178.628} C_VEL
LIN {X 0,Y 219.422,Z 445.975,A -85,B 0,C 180,E1 -23179.794,E2 -23179.794} C_VEL
LIN {X 0,Y 214.657,Z 434.356,A -85,B 0,C 180,E1 -23182.129,E2 -23182.129} C_VEL
LIN {X 0,Y 209.171,Z 422.803,A -85,B 0,C 180,E1 -23185.032,E2 -23185.032} C_VEL
LIN {X 0,Y 204.543,Z 414.168,A -85,B 0,C 180,E1 -23187.736,E2 -23187.736} C_VEL
LIN {X 0,Y 200.644,Z 407.237,A -85,B 0,C 180,E1 -23190.285,E2 -23190.285} C_VEL
LIN {X 0,Y 197.15,Z 401.657,A -85,B 0,C 180,E1 -23192.82,E2 -23192.82} C_VEL
LIN {X 0,Y 194.451,Z 397.662,A -85,B 0,C 180,E1 -23195.002,E2 -23195.002} C_VEL
LIN {X 0,Y 191.717,Z 394.416,A -85,B 0,C 180,E1 -23197.434,E2 -23197.434} C_VEL
LIN {X 0,Y 190.673,Z 392.722,A -85,B 0,C 180,E1 -23198.514,E2 -23198.514} C_VEL
LIN {X 0,Y 188.131,Z 390.17,A -85,B 0,C 180,E1 -23201.283,E2 -23201.283} C_VEL
LIN {X 0,Y 186.88,Z 387.667,A -85,B 0,C 180,E1 -23203.056,E2 -23203.056} C_VEL
LIN {X 0,Y 184.057,Z 385.361,A -85,B 0,C 180,E1 -23207.598,E2 -23207.598} C_VEL
LIN {X 0,Y 182.91,Z 382.557,A -85,B 0,C 180,E1 -23210.923,E2 -23210.923} C_VEL
LIN {X 0,Y 182.722,Z 381.972,A -85,B 0,C 180,E1 -23211.708,E2 -23211.708} C_VEL
LIN {X 0,Y 182.321,Z 381.751,A -85,B 0,C 180,E1 -23221.105,E2 -23221.105} C_VEL
LIN {X 0,Y 182.848,Z 382.099,A -85,B 0,C 180,E1 -23223.168,E2 -23223.168} C_VEL
LIN {X 0,Y 184.228,Z 385.253,A -85,B 0,C 180,E1 -23227.123,E2 -23227.123} C_VEL
LIN {X 0,Y 187.028,Z 387.832,A -85,B 0,C 180,E1 -23231.585,E2 -23231.585} C_VEL
LIN {X 0,Y 188.902,Z 391.062,A -85,B 0,C 180,E1 -23234.064,E2 -23234.064} C_VEL
LIN {X 0,Y 191.08,Z 393.264,A -85,B 0,C 180,E1 -23236.339,E2 -23236.339} C_VEL
LIN {X 0,Y 193.586,Z 396.835,A -85,B 0,C 180,E1 -23238.72,E2 -23238.72} C_VEL
LIN {X 0,Y 195.116,Z 398.613,A -85,B 0,C 180,E1 -23239.994,E2 -23239.994} C_VEL
LIN {X 0,Y 198.693,Z 403.516,A -85,B 0,C 180,E1 -23242.727,E2 -23242.727} C_VEL
LIN {X 0,Y 202.158,Z 408.451,A -85,B 0,C 180,E1 -23245.069,E2 -23245.069} C_VEL
LIN {X 0,Y 207.205,Z 415.978,A -85,B 0,C 180,E1 -23248.09,E2 -23248.09} C_VEL
LIN {X 0,Y 212.592,Z 424.836,A -85,B 0,C 180,E1 -23250.952,E2 -23250.952} C_VEL
LIN {X 0,Y 216.571,Z 432.112,A -85,B 0,C 180,E1 -23252.892,E2 -23252.892} C_VEL
LIN {X 0,Y 219.796,Z 439.348,A -85,B 0,C 180,E1 -23254.421,E2 -23254.421} C_VEL
LIN {X 0,Y 215.857,Z 491.357,A -85,B 0,C 180,E1 -23255.922,E2 -23255.922} C_VEL
LIN {X 0,Y 213.934,Z 504.954,A -85,B 0,C 180,E1 -23256.59,E2 -23256.59} C_VEL
LIN {X 0,Y 211.141,Z 518.627,A -85,B 0,C 180,E1 -23257.571,E2 -23257.571} C_VEL
LIN {X 0,Y 207.521,Z 531.837,A -85,B 0,C 180,E1 -23258.839,E2 -23258.839} C_VEL
LIN {X 0,Y 203.17,Z 544.57,A -85,B 0,C 180,E1 -23260.448,E2 -23260.448} C_VEL
LIN {X 0,Y 198.466,Z 556.194,A -85,B 0,C 180,E1 -23262.354,E2 -23262.354} C_VEL
LIN {X 0,Y 192.98,Z 567.709,A -85,B 0,C 180,E1 -23264.754,E2 -23264.754} C_VEL
LIN {X 0,Y 187.551,Z 578.003,A -85,B 0,C 180,E1 -23267.586,E2 -23267.586} C_VEL
LIN {X 0,Y 182.271,Z 587.036,A -85,B 0,C 180,E1 -23270.806,E2 -23270.806} C_VEL
LIN {X 0,Y 177.463,Z 594.568,A -85,B 0,C 180,E1 -23274.259,E2 -23274.259} C_VEL
LIN {X 0,Y 172.946,Z 601.044,A -85,B 0,C 180,E1 -23278.112,E2 -23278.112} C_VEL
LIN {X 0,Y 168.745,Z 606.76,A -85,B 0,C 180,E1 -23282.734,E2 -23282.734} C_VEL
LIN {X 0,Y 165.571,Z 610.886,A -85,B 0,C 180,E1 -23287.542,E2 -23287.542} C_VEL
LIN {X 0,Y 163.391,Z 613.551,A -85,B 0,C 180,E1 -23292.477,E2 -23292.477} C_VEL
LIN {X 0,Y 162.095,Z 614.838,A -85,B 0,C 180,E1 -23297.48,E2 -23297.48} C_VEL
LIN {X 0,Y 161.728,Z 614.778,A -85,B 0,C 180,E1 -23302.509,E2 -23302.509} C_VEL
LIN {X 0,Y 161.896,Z 613.662,A -85,B 0,C 180,E1 -23306.825,E2 -23306.825} C_VEL
LIN {X 0,Y 162.079,Z 612.206,A -85,B 0,C 180,E1 -23310,E2 -23310} C_VEL
LIN {X 0,Y 162.947,Z 608.801,A -85,B 0,C 180,E1 -23314.948,E2 -23314.948} C_VEL
LIN {X 0,Y 164.67,Z 603.923,A -85,B 0,C 180,E1 -23319.829,E2 -23319.829} C_VEL
LIN {X 0,Y 166.63,Z 599.213,A -85,B 0,C 180,E1 -23323.413,E2 -23323.413} C_VEL
LIN {X 0,Y 169.727,Z 592.044,A -85,B 0,C 180,E1 -23327.666,E2 -23327.666} C_VEL
LIN {X 0,Y 173.063,Z 583.954,A -85,B 0,C 180,E1 -23331.437,E2 -23331.437} C_VEL
LIN {X 0,Y 176.75,Z 575.132,A -85,B 0,C 180,E1 -23334.676,E2 -23334.676} C_VEL
LIN {X 0,Y 180.934,Z 564.451,A -85,B 0,C 180,E1 -23337.781,E2 -23337.781} C_VEL
LIN {X 0,Y 184.774,Z 553.636,A -85,B 0,C 180,E1 -23340.262,E2 -23340.262} C_VEL
LIN {X 0,Y 188.441,Z 541.8,A -85,B 0,C 180,E1 -23342.419,E2 -23342.419} C_VEL
LIN {X 0,Y 191.399,Z 530.483,A -85,B 0,C 180,E1 -23344.052,E2 -23344.052} C_VEL
LIN {X 0,Y 194.4,Z 517.233,A -85,B 0,C 180,E1 -23345.498,E2 -23345.498} C_VEL
LIN {X 0,Y 196.679,Z 503.593,A -85,B 0,C 180,E1 -23346.604,E2 -23346.604} C_VEL
LIN {X 0,Y 198.226,Z 489.632,A -85,B 0,C 180,E1 -23347.377,E2 -23347.377} C_VEL
LIN {X 0,Y 202.28,Z 423.821,A -85,B 0,C 180,E1 -23349.503,E2 -23349.503} C_VEL
LIN {X 0,Y 199.114,Z 416.333,A -85,B 0,C 180,E1 -23350.724,E2 -23350.724} C_VEL
LIN {X 0,Y 192.545,Z 404.046,A -85,B 0,C 180,E1 -23353.304,E2 -23353.304} C_VEL
LIN {X 0,Y 186.383,Z 394.104,A -85,B 0,C 180,E1 -23355.925,E2 -23355.925} C_VEL
LIN {X 0,Y 180.777,Z 385.925,A -85,B 0,C 180,E1 -23358.549,E2 -23358.549} C_VEL
LIN {X 0,Y 178.479,Z 382.748,A -85,B 0,C 180,E1 -23359.709,E2 -23359.709} C_VEL
LIN {X 0,Y 175.516,Z 378.679,A -85,B 0,C 180,E1 -23361.298,E2 -23361.298} C_VEL
LIN {X 0,Y 172.894,Z 375.199,A -85,B 0,C 180,E1 -23362.795,E2 -23362.795} C_VEL
LIN {X 0,Y 172.028,Z 374.104,A -85,B 0,C 180,E1 -23363.309,E2 -23363.309} C_VEL
LIN {X 0,Y 169.63,Z 371.44,A -85,B 0,C 180,E1 -23364.767,E2 -23364.767} C_VEL
LIN {X 0,Y 168.536,Z 369.262,A -85,B 0,C 180,E1 -23365.545,E2 -23365.545} C_VEL
LIN {X 0,Y 166.071,Z 367.462,A -85,B 0,C 180,E1 -23367.137,E2 -23367.137} C_VEL
LIN {X 0,Y 164.702,Z 365.043,A -85,B 0,C 180,E1 -23368.204,E2 -23368.204} C_VEL
LIN {X 0,Y 164.398,Z 363.63,A -85,B 0,C 180,E1 -23368.649,E2 -23368.649} C_VEL
LIN {X 0,Y 164.402,Z 363.619,A -85,B 0,C 180,E1 -23374.691,E2 -23374.691} C_VEL
LIN {X 0,Y 164.413,Z 363.6,A -85,B 0,C 180,E1 -23380.116,E2 -23380.116} C_VEL
LIN {X 0,Y 164.477,Z 363.603,A -85,B 0,C 180,E1 -23385.144,E2 -23385.144} C_VEL
LIN {X 0,Y 164.761,Z 363.576,A -85,B 0,C 180,E1 -23390.175,E2 -23390.175} C_VEL
LIN {X 0,Y 164.817,Z 363.569,A -85,B 0,C 180,E1 -23392.65,E2 -23392.65} C_VEL
LIN {X 0,Y 165.261,Z 363.525,A -85,B 0,C 180,E1 -23399.999,E2 -23399.999} C_VEL
LIN {X 0,Y 164.81,Z 363.574,A -85,B 0,C 180,E1 -23407.349,E2 -23407.349} C_VEL
LIN {X 0,Y 164.696,Z 363.581,A -85,B 0,C 180,E1 -23411.056,E2 -23411.056} C_VEL
LIN {X 0,Y 164.435,Z 363.617,A -85,B 0,C 180,E1 -23417.408,E2 -23417.408} C_VEL
LIN {X 0,Y 164.351,Z 363.625,A -85,B 0,C 180,E1 -23422.634,E2 -23422.634} C_VEL
LIN {X 0,Y 164.42,Z 363.771,A -85,B 0,C 180,E1 -23425.135,E2 -23425.135} C_VEL
LIN {X 0,Y 165.317,Z 366.378,A -85,B 0,C 180,E1 -23425.939,E2 -23425.939} C_VEL
LIN {X 0,Y 167.351,Z 368.592,A -85,B 0,C 180,E1 -23427.356,E2 -23427.356} C_VEL
LIN {X 0,Y 168.702,Z 369.466,A -85,B 0,C 180,E1 -23428.201,E2 -23428.201} C_VEL
LIN {X 0,Y 170.565,Z 372.646,A -85,B 0,C 180,E1 -23429.463,E2 -23429.463} C_VEL
LIN {X 0,Y 172.809,Z 374.896,A -85,B 0,C 180,E1 -23430.779,E2 -23430.779} C_VEL
LIN {X 0,Y 175.403,Z 378.519,A -85,B 0,C 180,E1 -23432.277,E2 -23432.277} C_VEL
LIN {X 0,Y 176.593,Z 380.015,A -85,B 0,C 180,E1 -23432.921,E2 -23432.921} C_VEL
LIN {X 0,Y 180.156,Z 385.033,A -85,B 0,C 180,E1 -23434.777,E2 -23434.777} C_VEL
LIN {X 0,Y 182.798,Z 388.854,A -85,B 0,C 180,E1 -23436.066,E2 -23436.066} C_VEL
LIN {X 0,Y 188.978,Z 400.155,A -85,B 0,C 180,E1 -23438.956,E2 -23438.956} C_VEL
LIN {X 0,Y 194.629,Z 412.02,A -85,B 0,C 180,E1 -23441.395,E2 -23441.395} C_VEL
LIN {X 0,Y 199.177,Z 423.245,A -85,B 0,C 180,E1 -23443.27,E2 -23443.27} C_VEL
LIN {X 0,Y 201.962,Z 430.887,A -85,B 0,C 180,E1 -23444.386,E2 -23444.386} C_VEL
LIN {X 0,Y 197.755,Z 497.957,A -85,B 0,C 180,E1 -23446.53,E2 -23446.53} C_VEL
LIN {X 0,Y 196.108,Z 511.824,A -85,B 0,C 180,E1 -23447.262,E2 -23447.262} C_VEL
LIN {X 0,Y 194.266,Z 522.644,A -85,B 0,C 180,E1 -23448.083,E2 -23448.083} C_VEL
LIN {X 0,Y 192.685,Z 528.188,A -85,B 0,C 180,E1 -23448.468,E2 -23448.468} C_VEL
LIN {X 0,Y 188.351,Z 537.013,A -85,B 0,C 180,E1 -23448.88,E2 -23448.88} C_VEL
LIN {X 0,Y 183.658,Z 545.544,A -85,B 0,C 180,E1 -23449.469,E2 -23449.469} C_VEL
LIN {X 0,Y 181.54,Z 550.627,A -85,B 0,C 180,E1 -23450.139,E2 -23450.139} C_VEL
LIN {X 0,Y 177.791,Z 561.998,A -85,B 0,C 180,E1 -23452.24,E2 -23452.24} C_VEL
LIN {X 0,Y 173.657,Z 572.927,A -85,B 0,C 180,E1 -23454.782,E2 -23454.782} C_VEL
LIN {X 0,Y 169.896,Z 582.146,A -85,B 0,C 180,E1 -23457.469,E2 -23457.469} C_VEL
LIN {X 0,Y 165.883,Z 591.383,A -85,B 0,C 180,E1 -23460.843,E2 -23460.843} C_VEL
LIN {X 0,Y 162.033,Z 600.21,A -85,B 0,C 180,E1 -23464.984,E2 -23464.984} C_VEL
LIN {X 0,Y 159.078,Z 607.336,A -85,B 0,C 180,E1 -23469.303,E2 -23469.303} C_VEL
LIN {X 0,Y 157.127,Z 612.283,A -85,B 0,C 180,E1 -23473.099,E2 -23473.099} C_VEL
LIN {X 0,Y 155.452,Z 617.382,A -85,B 0,C 180,E1 -23478.262,E2 -23478.262} C_VEL
LIN {X 0,Y 154.859,Z 620.223,A -85,B 0,C 180,E1 -23482.175,E2 -23482.175} C_VEL
LIN {X 0,Y 154.696,Z 622.707,A -85,B 0,C 180,E1 -23487.396,E2 -23487.396} C_VEL
LIN {X 0,Y 154.808,Z 623.432,A -85,B 0,C 180,E1 -23490,E2 -23490} C_VEL
LIN {X 0,Y 154.686,Z 623.852,A -85,B 0,C 180,E1 -23495.213,E2 -23495.213} C_VEL
LIN {X 0,Y 155.272,Z 622.946,A -85,B 0,C 180,E1 -23500.431,E2 -23500.431} C_VEL
LIN {X 0,Y 156.757,Z 620.71,A -85,B 0,C 180,E1 -23505.604,E2 -23505.604} C_VEL
LIN {X 0,Y 159.469,Z 617.094,A -85,B 0,C 180,E1 -23510.644,E2 -23510.644} C_VEL
LIN {X 0,Y 163.181,Z 611.995,A -85,B 0,C 180,E1 -23515.51,E2 -23515.51} C_VEL
LIN {X 0,Y 168.135,Z 605.261,A -85,B 0,C 180,E1 -23520.105,E2 -23520.105} C_VEL
LIN {X 0,Y 173.267,Z 597.773,A -85,B 0,C 180,E1 -23523.897,E2 -23523.897} C_VEL
LIN {X 0,Y 178.374,Z 589.987,A -85,B 0,C 180,E1 -23526.93,E2 -23526.93} C_VEL
LIN {X 0,Y 183.877,Z 580.625,A -85,B 0,C 180,E1 -23529.806,E2 -23529.806} C_VEL
LIN {X 0,Y 189.244,Z 570.282,A -85,B 0,C 180,E1 -23532.306,E2 -23532.306} C_VEL
LIN {X 0,Y 194.515,Z 558.896,A -85,B 0,C 180,E1 -23534.428,E2 -23534.428} C_VEL
LIN {X 0,Y 199.497,Z 546.307,A -85,B 0,C 180,E1 -23536.233,E2 -23536.233} C_VEL
LIN {X 0,Y 203.608,Z 534.089,A -85,B 0,C 180,E1 -23537.543,E2 -23537.543} C_VEL
LIN {X 0,Y 207.175,Z 520.619,A -85,B 0,C 180,E1 -23538.636,E2 -23538.636} C_VEL
LIN {X 0,Y 209.935,Z 506.741,A -85,B 0,C 180,E1 -23539.419,E2 -23539.419} C_VEL
LIN {X 0,Y 211.475,Z 494.173,A -85,B 0,C 180,E1 -23539.927,E2 -23539.927} C_VEL
LIN {X 0,Y 214.956,Z 448.49,A -85,B 0,C 180,E1 -23541.225,E2 -23541.225} C_VEL
LIN {X 0,Y 210.268,Z 436.959,A -85,B 0,C 180,E1 -23543.699,E2 -23543.699} C_VEL
LIN {X 0,Y 204.979,Z 425.757,A -85,B 0,C 180,E1 -23546.731,E2 -23546.731} C_VEL
LIN {X 0,Y 200.247,Z 416.699,A -85,B 0,C 180,E1 -23549.781,E2 -23549.781} C_VEL
LIN {X 0,Y 197.401,Z 411.784,A -85,B 0,C 180,E1 -23551.81,E2 -23551.81} C_VEL
LIN {X 0,Y 194.972,Z 407.736,A -85,B 0,C 180,E1 -23553.707,E2 -23553.707} C_VEL
LIN {X 0,Y 192.511,Z 404.027,A -85,B 0,C 180,E1 -23555.809,E2 -23555.809} C_VEL
LIN {X 0,Y 189.846,Z 400.564,A -85,B 0,C 180,E1 -23558.344,E2 -23558.344} C_VEL
LIN {X 0,Y 189.04,Z 399.366,A -85,B 0,C 180,E1 -23559.212,E2 -23559.212} C_VEL
LIN {X 0,Y 186.624,Z 396.673,A -85,B 0,C 180,E1 -23562.021,E2 -23562.021} C_VEL
LIN {X 0,Y 185.589,Z 394.552,A -85,B 0,C 180,E1 -23563.571,E2 -23563.571} C_VEL
LIN {X 0,Y 182.816,Z 392,A -85,B 0,C 180,E1 -23568.392,E2 -23568.392} C_VEL
LIN {X 0,Y 181.783,Z 389.001,A -85,B 0,C 180,E1 -23571.944,E2 -23571.944} C_VEL
LIN {X 0,Y 181.477,Z 388.792,A -85,B 0,C 180,E1 -23581.211,E2 -23581.211} C_VEL
LIN {X 0,Y 181.916,Z 389.311,A -85,B 0,C 180,E1 -23583.046,E2 -23583.046} C_VEL
LIN {X 0,Y 183.437,Z 392.548,A -85,B 0,C 180,E1 -23587.332,E2 -23587.332} C_VEL
LIN {X 0,Y 185.714,Z 394.702,A -85,B 0,C 180,E1 -23591.046,E2 -23591.046} C_VEL
LIN {X 0,Y 187.749,Z 398.051,A -85,B 0,C 180,E1 -23593.807,E2 -23593.807} C_VEL
LIN {X 0,Y 189.523,Z 399.949,A -85,B 0,C 180,E1 -23595.735,E2 -23595.735} C_VEL
LIN {X 0,Y 192.078,Z 403.605,A -85,B 0,C 180,E1 -23598.254,E2 -23598.254} C_VEL
LIN {X 0,Y 193.285,Z 405.137,A -85,B 0,C 180,E1 -23599.309,E2 -23599.309} C_VEL
LIN {X 0,Y 196.677,Z 409.87,A -85,B 0,C 180,E1 -23602.021,E2 -23602.021} C_VEL
LIN {X 0,Y 200.16,Z 415.042,A -85,B 0,C 180,E1 -23604.482,E2 -23604.482} C_VEL
LIN {X 0,Y 205.006,Z 422.488,A -85,B 0,C 180,E1 -23607.497,E2 -23607.497} C_VEL
LIN {X 0,Y 210.1,Z 431.305,A -85,B 0,C 180,E1 -23610.325,E2 -23610.325} C_VEL
LIN {X 0,Y 213.19,Z 437.195,A -85,B 0,C 180,E1 -23611.911,E2 -23611.911} C_VEL
LIN {X 0,Y 215.4,Z 442.27,A -85,B 0,C 180,E1 -23613.028,E2 -23613.028} C_VEL
LIN {X 0,Y 211.507,Z 491.121,A -85,B 0,C 180,E1 -23614.413,E2 -23614.413} C_VEL
LIN {X 0,Y 209.522,Z 504.846,A -85,B 0,C 180,E1 -23615.08,E2 -23615.08} C_VEL
LIN {X 0,Y 206.556,Z 518.939,A -85,B 0,C 180,E1 -23616.093,E2 -23616.093} C_VEL
LIN {X 0,Y 202.533,Z 533.017,A -85,B 0,C 180,E1 -23617.463,E2 -23617.463} C_VEL
LIN {X 0,Y 198.048,Z 545.562,A -85,B 0,C 180,E1 -23619.082,E2 -23619.082} C_VEL
LIN {X 0,Y 192.866,Z 557.656,A -85,B 0,C 180,E1 -23621.103,E2 -23621.103} C_VEL
LIN {X 0,Y 187.99,Z 567.466,A -85,B 0,C 180,E1 -23623.199,E2 -23623.199} C_VEL
LIN {X 0,Y 183.204,Z 576.233,A -85,B 0,C 180,E1 -23625.567,E2 -23625.567} C_VEL
LIN {X 0,Y 177.566,Z 585.587,A -85,B 0,C 180,E1 -23628.767,E2 -23628.767} C_VEL
LIN {X 0,Y 172.37,Z 593.498,A -85,B 0,C 180,E1 -23632.296,E2 -23632.296} C_VEL
LIN {X 0,Y 168.123,Z 599.347,A -85,B 0,C 180,E1 -23635.645,E2 -23635.645} C_VEL
LIN {X 0,Y 164.445,Z 604.152,A -85,B 0,C 180,E1 -23639.147,E2 -23639.147} C_VEL
LIN {X 0,Y 160.489,Z 609.095,A -85,B 0,C 180,E1 -23644.03,E2 -23644.03} C_VEL
LIN {X 0,Y 157.613,Z 612.515,A -85,B 0,C 180,E1 -23649.102,E2 -23649.102} C_VEL
LIN {X 0,Y 155.697,Z 614.523,A -85,B 0,C 180,E1 -23654.287,E2 -23654.287} C_VEL
LIN {X 0,Y 154.776,Z 615.178,A -85,B 0,C 180,E1 -23659.536,E2 -23659.536} C_VEL
LIN {X 0,Y 154.717,Z 614.495,A -85,B 0,C 180,E1 -23664.788,E2 -23664.788} C_VEL
LIN {X 0,Y 154.819,Z 613.658,A -85,B 0,C 180,E1 -23667.398,E2 -23667.398} C_VEL
LIN {X 0,Y 155.381,Z 610.98,A -85,B 0,C 180,E1 -23672.592,E2 -23672.592} C_VEL
LIN {X 0,Y 156.684,Z 606.897,A -85,B 0,C 180,E1 -23677.733,E2 -23677.733} C_VEL
LIN {X 0,Y 158.985,Z 601.27,A -85,B 0,C 180,E1 -23682.769,E2 -23682.769} C_VEL
LIN {X 0,Y 161.597,Z 595.678,A -85,B 0,C 180,E1 -23686.575,E2 -23686.575} C_VEL
LIN {X 0,Y 164.932,Z 588.26,A -85,B 0,C 180,E1 -23690.581,E2 -23690.581} C_VEL
LIN {X 0,Y 168.381,Z 580.283,A -85,B 0,C 180,E1 -23694.013,E2 -23694.013} C_VEL
LIN {X 0,Y 172.431,Z 570.661,A -85,B 0,C 180,E1 -23697.291,E2 -23697.291} C_VEL
LIN {X 0,Y 176.637,Z 559.983,A -85,B 0,C 180,E1 -23700.153,E2 -23700.153} C_VEL
LIN {X 0,Y 180.762,Z 548.16,A -85,B 0,C 180,E1 -23702.646,E2 -23702.646} C_VEL
LIN {X 0,Y 184.197,Z 536.561,A -85,B 0,C 180,E1 -23704.579,E2 -23704.579} C_VEL
LIN {X 0,Y 187.706,Z 522.91,A -85,B 0,C 180,E1 -23706.301,E2 -23706.301} C_VEL
LIN {X 0,Y 190.469,Z 508.945,A -85,B 0,C 180,E1 -23707.587,E2 -23707.587} C_VEL
LIN {X 0,Y 192.385,Z 495.223,A -85,B 0,C 180,E1 -23708.474,E2 -23708.474} C_VEL
LIN {X 0,Y 193.656,Z 479.724,A -85,B 0,C 180,E1 -23709.099,E2 -23709.099} C_VEL
LIN {X 0,Y 196.962,Z 425.877,A -85,B 0,C 180,E1 -23710.856,E2 -23710.856} C_VEL
LIN {X 0,Y 194.327,Z 419.713,A -85,B 0,C 180,E1 -23711.935,E2 -23711.935} C_VEL
LIN {X 0,Y 187.669,Z 407.228,A -85,B 0,C 180,E1 -23714.728,E2 -23714.728} C_VEL
LIN {X 0,Y 181.174,Z 396.731,A -85,B 0,C 180,E1 -23717.716,E2 -23717.716} C_VEL
LIN {X 0,Y 175.612,Z 388.703,A -85,B 0,C 180,E1 -23720.565,E2 -23720.565} C_VEL
LIN {X 0,Y 172.352,Z 384.205,A -85,B 0,C 180,E1 -23722.405,E2 -23722.405} C_VEL
LIN {X 0,Y 169.498,Z 380.293,A -85,B 0,C 180,E1 -23724.148,E2 -23724.148} C_VEL
LIN {X 0,Y 166.894,Z 377.197,A -85,B 0,C 180,E1 -23725.831,E2 -23725.831} C_VEL
LIN {X 0,Y 165.862,Z 375.528,A -85,B 0,C 180,E1 -23726.574,E2 -23726.574} C_VEL
LIN {X 0,Y 163.427,Z 373.179,A -85,B 0,C 180,E1 -23728.292,E2 -23728.292} C_VEL
LIN {X 0,Y 161.845,Z 370.268,A -85,B 0,C 180,E1 -23729.623,E2 -23729.623} C_VEL
LIN {X 0,Y 159.26,Z 368.58,A -85,B 0,C 180,E1 -23731.68,E2 -23731.68} C_VEL
LIN {X 0,Y 157.751,Z 366.215,A -85,B 0,C 180,E1 -23733.143,E2 -23733.143} C_VEL
LIN {X 0,Y 157.336,Z 364.489,A -85,B 0,C 180,E1 -23733.762,E2 -23733.762} C_VEL
LIN {X 0,Y 157.357,Z 364.478,A -85,B 0,C 180,E1 -23739.701,E2 -23739.701} C_VEL
LIN {X 0,Y 157.409,Z 364.493,A -85,B 0,C 180,E1 -23744.46,E2 -23744.46} C_VEL
LIN {X 0,Y 157.683,Z 364.45,A -85,B 0,C 180,E1 -23749.729,E2 -23749.729} C_VEL
LIN {X 0,Y 157.755,Z 364.453,A -85,B 0,C 180,E1 -23752.319,E2 -23752.319} C_VEL
LIN {X 0,Y 158.224,Z 364.401,A -85,B 0,C 180,E1 -23759.999,E2 -23759.999} C_VEL
LIN {X 0,Y 157.749,Z 364.449,A -85,B 0,C 180,E1 -23767.68,E2 -23767.68} C_VEL
LIN {X 0,Y 157.627,Z 364.462,A -85,B 0,C 180,E1 -23771.225,E2 -23771.225} C_VEL
LIN {X 0,Y 157.412,Z 364.482,A -85,B 0,C 180,E1 -23775.537,E2 -23775.537} C_VEL
LIN {X 0,Y 157.378,Z 364.518,A -85,B 0,C 180,E1 -23779.991,E2 -23779.991} C_VEL
LIN {X 0,Y 158.018,Z 366.809,A -85,B 0,C 180,E1 -23780.783,E2 -23780.783} C_VEL
LIN {X 0,Y 159.84,Z 369.111,A -85,B 0,C 180,E1 -23782.456,E2 -23782.456} C_VEL
LIN {X 0,Y 162.024,Z 370.548,A -85,B 0,C 180,E1 -23784.164,E2 -23784.164} C_VEL
LIN {X 0,Y 163.678,Z 373.535,A -85,B 0,C 180,E1 -23785.537,E2 -23785.537} C_VEL
LIN {X 0,Y 166.328,Z 376.069,A -85,B 0,C 180,E1 -23787.382,E2 -23787.382} C_VEL
LIN {X 0,Y 168.696,Z 379.483,A -85,B 0,C 180,E1 -23788.995,E2 -23788.995} C_VEL
LIN {X 0,Y 170.266,Z 381.238,A -85,B 0,C 180,E1 -23789.964,E2 -23789.964} C_VEL
LIN {X 0,Y 174.145,Z 386.601,A -85,B 0,C 180,E1 -23792.258,E2 -23792.258} C_VEL
LIN {X 0,Y 179.112,Z 393.655,A -85,B 0,C 180,E1 -23794.899,E2 -23794.899} C_VEL
LIN {X 0,Y 185.037,Z 404.841,A -85,B 0,C 180,E1 -23797.852,E2 -23797.852} C_VEL
LIN {X 0,Y 189.903,Z 415.307,A -85,B 0,C 180,E1 -23800.096,E2 -23800.096} C_VEL
LIN {X 0,Y 194.056,Z 425.601,A -85,B 0,C 180,E1 -23801.925,E2 -23801.925} C_VEL
LIN {X 0,Y 196.665,Z 432.889,A -85,B 0,C 180,E1 -23803.047,E2 -23803.047} C_VEL
LIN {X 0,Y 192.391,Z 498.327,A -85,B 0,C 180,E1 -23805.179,E2 -23805.179} C_VEL
LIN {X 0,Y 190.527,Z 512.744,A -85,B 0,C 180,E1 -23805.967,E2 -23805.967} C_VEL
LIN {X 0,Y 187.885,Z 526.91,A -85,B 0,C 180,E1 -23807.133,E2 -23807.133} C_VEL
LIN {X 0,Y 184.644,Z 540.018,A -85,B 0,C 180,E1 -23808.6,E2 -23808.6} C_VEL
LIN {X 0,Y 181.54,Z 550.627,A -85,B 0,C 180,E1 -23810.139,E2 -23810.139} C_VEL
LIN {X 0,Y 179.366,Z 555.702,A -85,B 0,C 180,E1 -23810.883,E2 -23810.883} C_VEL
LIN {X 0,Y 174.19,Z 563.601,A -85,B 0,C 180,E1 -23811.92,E2 -23811.92} C_VEL
LIN {X 0,Y 168.943,Z 571.083,A -85,B 0,C 180,E1 -23813.155,E2 -23813.155} C_VEL
LIN {X 0,Y 166.624,Z 575.434,A -85,B 0,C 180,E1 -23814.234,E2 -23814.234} C_VEL
LIN {X 0,Y 162.4,Z 584.911,A -85,B 0,C 180,E1 -23817.253,E2 -23817.253} C_VEL
LIN {X 0,Y 158.399,Z 593.654,A -85,B 0,C 180,E1 -23820.788,E2 -23820.788} C_VEL
LIN {X 0,Y 154.562,Z 602.032,A -85,B 0,C 180,E1 -23825.128,E2 -23825.128} C_VEL
LIN {X 0,Y 151.624,Z 608.755,A -85,B 0,C 180,E1 -23829.658,E2 -23829.658} C_VEL
LIN {X 0,Y 149.685,Z 613.382,A -85,B 0,C 180,E1 -23833.638,E2 -23833.638} C_VEL
LIN {X 0,Y 148.207,Z 618.151,A -85,B 0,C 180,E1 -23839.066,E2 -23839.066} C_VEL
LIN {X 0,Y 147.624,Z 621.384,A -85,B 0,C 180,E1 -23844.537,E2 -23844.537} C_VEL
LIN {X 0,Y 147.715,Z 623.208,A -85,B 0,C 180,E1 -23850,E2 -23850} C_VEL
LIN {X 0,Y 147.606,Z 623.6,A -85,B 0,C 180,E1 -23852.729,E2 -23852.729} C_VEL
LIN {X 0,Y 147.805,Z 623.385,A -85,B 0,C 180,E1 -23858.201,E2 -23858.201} C_VEL
LIN {X 0,Y 148.944,Z 621.848,A -85,B 0,C 180,E1 -23863.646,E2 -23863.646} C_VEL
LIN {X 0,Y 151.24,Z 618.965,A -85,B 0,C 180,E1 -23868.982,E2 -23868.982} C_VEL
LIN {X 0,Y 154.672,Z 614.656,A -85,B 0,C 180,E1 -23874.138,E2 -23874.138} C_VEL
LIN {X 0,Y 159.234,Z 608.801,A -85,B 0,C 180,E1 -23879.044,E2 -23879.044} C_VEL
LIN {X 0,Y 164.21,Z 602.233,A -85,B 0,C 180,E1 -23883.07,E2 -23883.07} C_VEL
LIN {X 0,Y 169.981,Z 594.109,A -85,B 0,C 180,E1 -23886.834,E2 -23886.834} C_VEL
LIN {X 0,Y 175.542,Z 585.625,A -85,B 0,C 180,E1 -23889.834,E2 -23889.834} C_VEL
LIN {X 0,Y 181.456,Z 575.37,A -85,B 0,C 180,E1 -23892.678,E2 -23892.678} C_VEL
LIN {X 0,Y 187.329,Z 563.953,A -85,B 0,C 180,E1 -23895.081,E2 -23895.081} C_VEL
LIN {X 0,Y 192.363,Z 552.586,A -85,B 0,C 180,E1 -23896.944,E2 -23896.944} C_VEL
LIN {X 0,Y 197.1,Z 540.148,A -85,B 0,C 180,E1 -23898.484,E2 -23898.484} C_VEL
LIN {X 0,Y 201.35,Z 526.254,A -85,B 0,C 180,E1 -23899.775,E2 -23899.775} C_VEL
LIN {X 0,Y 204.593,Z 512.254,A -85,B 0,C 180,E1 -23900.71,E2 -23900.71} C_VEL
LIN {X 0,Y 206.871,Z 497.535,A -85,B 0,C 180,E1 -23901.385,E2 -23901.385} C_VEL
LIN {X 0,Y 210.624,Z 451.07,A -85,B 0,C 180,E1 -23902.716,E2 -23902.716} C_VEL
LIN {X 0,Y 206.288,Z 440.322,A -85,B 0,C 180,E1 -23905.178,E2 -23905.178} C_VEL
LIN {X 0,Y 201.668,Z 430.278,A -85,B 0,C 180,E1 -23908.034,E2 -23908.034} C_VEL
LIN {X 0,Y 197.284,Z 421.608,A -85,B 0,C 180,E1 -23911.077,E2 -23911.077} C_VEL
LIN {X 0,Y 193.492,Z 414.794,A -85,B 0,C 180,E1 -23914.07,E2 -23914.07} C_VEL
LIN {X 0,Y 190.663,Z 410.445,A -85,B 0,C 180,E1 -23916.585,E2 -23916.585} C_VEL
LIN {X 0,Y 188.028,Z 406.74,A -85,B 0,C 180,E1 -23919.266,E2 -23919.266} C_VEL
LIN {X 0,Y 186.741,Z 405.307,A -85,B 0,C 180,E1 -23920.708,E2 -23920.708} C_VEL
LIN {X 0,Y 184.471,Z 401.83,A -85,B 0,C 180,E1 -23923.824,E2 -23923.824} C_VEL
LIN {X 0,Y 184.045,Z 401.214,A -85,B 0,C 180,E1 -23924.497,E2 -23924.497} C_VEL
LIN {X 0,Y 181.525,Z 398.429,A -85,B 0,C 180,E1 -23929.447,E2 -23929.447} C_VEL
LIN {X 0,Y 180.828,Z 396.025,A -85,B 0,C 180,E1 -23932.253,E2 -23932.253} C_VEL
LIN {X 0,Y 180.609,Z 395.841,A -85,B 0,C 180,E1 -23941.217,E2 -23941.217} C_VEL
LIN {X 0,Y 180.932,Z 396.254,A -85,B 0,C 180,E1 -23942.645,E2 -23942.645} C_VEL
LIN {X 0,Y 182.476,Z 399.606,A -85,B 0,C 180,E1 -23947.192,E2 -23947.192} C_VEL
LIN {X 0,Y 184.467,Z 401.633,A -85,B 0,C 180,E1 -23950.574,E2 -23950.574} C_VEL
LIN {X 0,Y 186.651,Z 405.129,A -85,B 0,C 180,E1 -23953.612,E2 -23953.612} C_VEL
LIN {X 0,Y 188.028,Z 406.717,A -85,B 0,C 180,E1 -23955.168,E2 -23955.168} C_VEL
LIN {X 0,Y 190.653,Z 410.449,A -85,B 0,C 180,E1 -23957.845,E2 -23957.845} C_VEL
LIN {X 0,Y 194.69,Z 416.242,A -85,B 0,C 180,E1 -23961.3,E2 -23961.3} C_VEL
LIN {X 0,Y 198.933,Z 422.677,A -85,B 0,C 180,E1 -23964.388,E2 -23964.388} C_VEL
LIN {X 0,Y 204.418,Z 431.792,A -85,B 0,C 180,E1 -23967.848,E2 -23967.848} C_VEL
LIN {X 0,Y 209.515,Z 441.407,A -85,B 0,C 180,E1 -23970.699,E2 -23970.699} C_VEL
LIN {X 0,Y 211.04,Z 444.92,A -85,B 0,C 180,E1 -23971.523,E2 -23971.523} C_VEL
LIN {X 0,Y 207.221,Z 491.614,A -85,B 0,C 180,E1 -23972.872,E2 -23972.872} C_VEL
LIN {X 0,Y 205.174,Z 505.213,A -85,B 0,C 180,E1 -23973.535,E2 -23973.535} C_VEL
LIN {X 0,Y 202.11,Z 519.258,A -85,B 0,C 180,E1 -23974.547,E2 -23974.547} C_VEL
LIN {X 0,Y 198.239,Z 532.416,A -85,B 0,C 180,E1 -23975.812,E2 -23975.812} C_VEL
LIN {X 0,Y 193.582,Z 545.114,A -85,B 0,C 180,E1 -23977.425,E2 -23977.425} C_VEL
LIN {X 0,Y 188.23,Z 557.324,A -85,B 0,C 180,E1 -23979.458,E2 -23979.458} C_VEL
LIN {X 0,Y 183.156,Z 567.224,A -85,B 0,C 180,E1 -23981.563,E2 -23981.563} C_VEL
LIN {X 0,Y 178.103,Z 576.063,A -85,B 0,C 180,E1 -23983.935,E2 -23983.935} C_VEL
LIN {X 0,Y 172.601,Z 584.859,A -85,B 0,C 180,E1 -23986.942,E2 -23986.942} C_VEL
LIN {X 0,Y 167.517,Z 592.326,A -85,B 0,C 180,E1 -23990.224,E2 -23990.224} C_VEL
LIN {X 0,Y 162.203,Z 599.345,A -85,B 0,C 180,E1 -23994.203,E2 -23994.203} C_VEL
LIN {X 0,Y 158.29,Z 604.193,A -85,B 0,C 180,E1 -23997.807,E2 -23997.807} C_VEL
LIN {X 0,Y 154.008,Z 609.178,A -85,B 0,C 180,E1 -24002.85,E2 -24002.85} C_VEL
LIN {X 0,Y 150.874,Z 612.637,A -85,B 0,C 180,E1 -24008.121,E2 -24008.121} C_VEL
LIN {X 0,Y 148.791,Z 614.681,A -85,B 0,C 180,E1 -24013.537,E2 -24013.537} C_VEL
LIN {X 0,Y 147.711,Z 615.376,A -85,B 0,C 180,E1 -24019.029,E2 -24019.029} C_VEL
LIN {X 0,Y 147.615,Z 614.737,A -85,B 0,C 180,E1 -24024.536,E2 -24024.536} C_VEL
LIN {X 0,Y 147.729,Z 613.82,A -85,B 0,C 180,E1 -24027.524,E2 -24027.524} C_VEL
LIN {X 0,Y 148.29,Z 611.283,A -85,B 0,C 180,E1 -24032.716,E2 -24032.716} C_VEL
LIN {X 0,Y 149.675,Z 607.237,A -85,B 0,C 180,E1 -24038.098,E2 -24038.098} C_VEL
LIN {X 0,Y 152.08,Z 601.653,A -85,B 0,C 180,E1 -24043.359,E2 -24043.359} C_VEL
LIN {X 0,Y 155.057,Z 595.554,A -85,B 0,C 180,E1 -24047.673,E2 -24047.673} C_VEL
LIN {X 0,Y 158.852,Z 587.521,A -85,B 0,C 180,E1 -24052.089,E2 -24052.089} C_VEL
LIN {X 0,Y 162.629,Z 579.342,A -85,B 0,C 180,E1 -24055.603,E2 -24055.603} C_VEL
LIN {X 0,Y 166.981,Z 569.49,A -85,B 0,C 180,E1 -24058.947,E2 -24058.947} C_VEL
LIN {X 0,Y 171.406,Z 558.54,A -85,B 0,C 180,E1 -24061.863,E2 -24061.863} C_VEL
LIN {X 0,Y 175.784,Z 546.313,A -85,B 0,C 180,E1 -24064.382,E2 -24064.382} C_VEL
LIN {X 0,Y 179.364,Z 534.23,A -85,B 0,C 180,E1 -24066.343,E2 -24066.343} C_VEL
LIN {X 0,Y 182.844,Z 520.787,A -85,B 0,C 180,E1 -24067.95,E2 -24067.95} C_VEL
LIN {X 0,Y 185.564,Z 506.73,A -85,B 0,C 180,E1 -24069.198,E2 -24069.198} C_VEL
LIN {X 0,Y 187.382,Z 492.774,A -85,B 0,C 180,E1 -24070.066,E2 -24070.066} C_VEL
LIN {X 0,Y 189.031,Z 470.915,A -85,B 0,C 180,E1 -24070.855,E2 -24070.855} C_VEL
LIN {X 0,Y 191.737,Z 427.826,A -85,B 0,C 180,E1 -24072.296,E2 -24072.296} C_VEL
LIN {X 0,Y 186.177,Z 416.398,A -85,B 0,C 180,E1 -24074.72,E2 -24074.72} C_VEL
LIN {X 0,Y 179.832,Z 405.353,A -85,B 0,C 180,E1 -24077.708,E2 -24077.708} C_VEL
LIN {X 0,Y 173.234,Z 395.176,A -85,B 0,C 180,E1 -24081.203,E2 -24081.203} C_VEL
LIN {X 0,Y 169.381,Z 389.883,A -85,B 0,C 180,E1 -24083.475,E2 -24083.475} C_VEL
LIN {X 0,Y 166.641,Z 386.116,A -85,B 0,C 180,E1 -24085.247,E2 -24085.247} C_VEL
LIN {X 0,Y 163.919,Z 382.419,A -85,B 0,C 180,E1 -24087.16,E2 -24087.16} C_VEL
LIN {X 0,Y 160.701,Z 378.708,A -85,B 0,C 180,E1 -24089.609,E2 -24089.609} C_VEL
LIN {X 0,Y 159.732,Z 376.837,A -85,B 0,C 180,E1 -24090.483,E2 -24090.483} C_VEL
LIN {X 0,Y 157.099,Z 374.748,A -85,B 0,C 180,E1 -24092.735,E2 -24092.735} C_VEL
LIN {X 0,Y 155.456,Z 371.88,A -85,B 0,C 180,E1 -24094.476,E2 -24094.476} C_VEL
LIN {X 0,Y 155.083,Z 371.227,A -85,B 0,C 180,E1 -24094.894,E2 -24094.894} C_VEL
LIN {X 0,Y 152.252,Z 369.53,A -85,B 0,C 180,E1 -24097.971,E2 -24097.971} C_VEL
LIN {X 0,Y 150.696,Z 366.96,A -85,B 0,C 180,E1 -24100.214,E2 -24100.214} C_VEL
LIN {X 0,Y 150.303,Z 365.361,A -85,B 0,C 180,E1 -24101.07,E2 -24101.07} C_VEL
LIN {X 0,Y 150.404,Z 365.342,A -85,B 0,C 180,E1 -24106.488,E2 -24106.488} C_VEL
LIN {X 0,Y 150.602,Z 365.325,A -85,B 0,C 180,E1 -24109.241,E2 -24109.241} C_VEL
LIN {X 0,Y 150.694,Z 365.336,A -85,B 0,C 180,E1 -24111.956,E2 -24111.956} C_VEL
LIN {X 0,Y 151.184,Z 365.278,A -85,B 0,C 180,E1 -24119.999,E2 -24119.999} C_VEL
LIN {X 0,Y 150.673,Z 365.326,A -85,B 0,C 180,E1 -24128.043,E2 -24128.043} C_VEL
LIN {X 0,Y 150.464,Z 365.373,A -85,B 0,C 180,E1 -24132.856,E2 -24132.856} C_VEL
LIN {X 0,Y 151.046,Z 367.603,A -85,B 0,C 180,E1 -24133.966,E2 -24133.966} C_VEL
LIN {X 0,Y 152.969,Z 370.056,A -85,B 0,C 180,E1 -24136.515,E2 -24136.515} C_VEL
LIN {X 0,Y 155.405,Z 371.585,A -85,B 0,C 180,E1 -24139.083,E2 -24139.083} C_VEL
LIN {X 0,Y 156.679,Z 374.207,A -85,B 0,C 180,E1 -24140.496,E2 -24140.496} C_VEL
LIN {X 0,Y 159.187,Z 376.537,A -85,B 0,C 180,E1 -24142.724,E2 -24142.724} C_VEL
LIN {X 0,Y 159.889,Z 377.17,A -85,B 0,C 180,E1 -24143.303,E2 -24143.303} C_VEL
LIN {X 0,Y 162.132,Z 380.575,A -85,B 0,C 180,E1 -24145.172,E2 -24145.172} C_VEL
LIN {X 0,Y 164.044,Z 382.537,A -85,B 0,C 180,E1 -24146.561,E2 -24146.561} C_VEL
LIN {X 0,Y 166.788,Z 386.218,A -85,B 0,C 180,E1 -24148.479,E2 -24148.479} C_VEL
LIN {X 0,Y 171.252,Z 392.395,A -85,B 0,C 180,E1 -24151.291,E2 -24151.291} C_VEL
LIN {X 0,Y 175.807,Z 399.088,A -85,B 0,C 180,E1 -24153.859,E2 -24153.859} C_VEL
LIN {X 0,Y 181.454,Z 410.128,A -85,B 0,C 180,E1 -24156.847,E2 -24156.847} C_VEL
LIN {X 0,Y 186.503,Z 421.448,A -85,B 0,C 180,E1 -24159.312,E2 -24159.312} C_VEL
LIN {X 0,Y 191.295,Z 434.329,A -85,B 0,C 180,E1 -24161.548,E2 -24161.548} C_VEL
LIN {X 0,Y 191.458,Z 436.217,A -85,B 0,C 180,E1 -24161.697,E2 -24161.697} C_VEL
LIN {X 0,Y 187.144,Z 498.425,A -85,B 0,C 180,E1 -24163.735,E2 -24163.735} C_VEL
LIN {X 0,Y 185.199,Z 512.889,A -85,B 0,C 180,E1 -24164.545,E2 -24164.545} C_VEL
LIN {X 0,Y 182.458,Z 526.965,A -85,B 0,C 180,E1 -24165.723,E2 -24165.723} C_VEL
LIN {X 0,Y 179.366,Z 539.13,A -85,B 0,C 180,E1 -24167.096,E2 -24167.096} C_VEL
LIN {X 0,Y 175.42,Z 551.953,A -85,B 0,C 180,E1 -24169.002,E2 -24169.002} C_VEL
LIN {X 0,Y 171.144,Z 564.28,A -85,B 0,C 180,E1 -24171.434,E2 -24171.434} C_VEL
LIN {X 0,Y 167.065,Z 574.316,A -85,B 0,C 180,E1 -24173.919,E2 -24173.919} C_VEL
LIN {X 0,Y 166.624,Z 575.434,A -85,B 0,C 180,E1 -24174.234,E2 -24174.234} C_VEL
LIN {X 0,Y 164.295,Z 579.71,A -85,B 0,C 180,E1 -24175.391,E2 -24175.391} C_VEL
LIN {X 0,Y 158.799,Z 586.288,A -85,B 0,C 180,E1 -24177.16,E2 -24177.16} C_VEL
LIN {X 0,Y 153.255,Z 592.362,A -85,B 0,C 180,E1 -24179.203,E2 -24179.203} C_VEL
LIN {X 0,Y 150.917,Z 595.838,A -85,B 0,C 180,E1 -24180.773,E2 -24180.773} C_VEL
LIN {X 0,Y 147.144,Z 603.487,A -85,B 0,C 180,E1 -24185.159,E2 -24185.159} C_VEL
LIN {X 0,Y 144.199,Z 610.03,A -85,B 0,C 180,E1 -24190.053,E2 -24190.053} C_VEL
LIN {X 0,Y 141.854,Z 615.641,A -85,B 0,C 180,E1 -24195.658,E2 -24195.658} C_VEL
LIN {X 0,Y 140.754,Z 619.672,A -85,B 0,C 180,E1 -24201.385,E2 -24201.385} C_VEL
LIN {X 0,Y 140.503,Z 622.227,A -85,B 0,C 180,E1 -24207.133,E2 -24207.133} C_VEL
LIN {X 0,Y 140.567,Z 623.088,A -85,B 0,C 180,E1 -24210.644,E2 -24210.644} C_VEL
LIN {X 0,Y 140.532,Z 623.464,A -85,B 0,C 180,E1 -24215.74,E2 -24215.74} C_VEL
LIN {X 0,Y 141.253,Z 622.618,A -85,B 0,C 180,E1 -24221.479,E2 -24221.479} C_VEL
LIN {X 0,Y 143.045,Z 620.445,A -85,B 0,C 180,E1 -24227.144,E2 -24227.144} C_VEL
LIN {X 0,Y 146.183,Z 616.896,A -85,B 0,C 180,E1 -24232.619,E2 -24232.619} C_VEL
LIN {X 0,Y 150.417,Z 611.866,A -85,B 0,C 180,E1 -24237.854,E2 -24237.854} C_VEL
LIN {X 0,Y 155.944,Z 605.215,A -85,B 0,C 180,E1 -24242.738,E2 -24242.738} C_VEL
LIN {X 0,Y 161.624,Z 597.835,A -85,B 0,C 180,E1 -24246.719,E2 -24246.719} C_VEL
LIN {X 0,Y 168.183,Z 588.682,A -85,B 0,C 180,E1 -24250.368,E2 -24250.368} C_VEL
LIN {X 0,Y 174.214,Z 579.137,A -85,B 0,C 180,E1 -24253.297,E2 -24253.297} C_VEL
LIN {X 0,Y 180.097,Z 568.579,A -85,B 0,C 180,E1 -24255.81,E2 -24255.81} C_VEL
LIN {X 0,Y 185.798,Z 556.928,A -85,B 0,C 180,E1 -24257.929,E2 -24257.929} C_VEL
LIN {X 0,Y 190.627,Z 545.558,A -85,B 0,C 180,E1 -24259.497,E2 -24259.497} C_VEL
LIN {X 0,Y 194.962,Z 533.258,A -85,B 0,C 180,E1 -24260.806,E2 -24260.806} C_VEL
LIN {X 0,Y 198.752,Z 519.659,A -85,B 0,C 180,E1 -24261.883,E2 -24261.883} C_VEL
LIN {X 0,Y 201.639,Z 505.567,A -85,B 0,C 180,E1 -24262.664,E2 -24262.664} C_VEL
LIN {X 0,Y 203.425,Z 491.401,A -85,B 0,C 180,E1 -24263.189,E2 -24263.189} C_VEL
LIN {X 0,Y 206.423,Z 453.751,A -85,B 0,C 180,E1 -24264.27,E2 -24264.27} C_VEL
LIN {X 0,Y 202.52,Z 443.807,A -85,B 0,C 180,E1 -24266.673,E2 -24266.673} C_VEL
LIN {X 0,Y 198.053,Z 433.842,A -85,B 0,C 180,E1 -24269.678,E2 -24269.678} C_VEL
LIN {X 0,Y 193.884,Z 425.394,A -85,B 0,C 180,E1 -24272.857,E2 -24272.857} C_VEL
LIN {X 0,Y 190.586,Z 419.51,A -85,B 0,C 180,E1 -24275.717,E2 -24275.717} C_VEL
LIN {X 0,Y 189.029,Z 417.041,A -85,B 0,C 180,E1 -24277.208,E2 -24277.208} C_VEL
LIN {X 0,Y 186.35,Z 413.085,A -85,B 0,C 180,E1 -24280.094,E2 -24280.094} C_VEL
LIN {X 0,Y 183.676,Z 409.645,A -85,B 0,C 180,E1 -24283.574,E2 -24283.574} C_VEL
LIN {X 0,Y 183.024,Z 408.193,A -85,B 0,C 180,E1 -24284.693,E2 -24284.693} C_VEL
LIN {X 0,Y 180.587,Z 405.524,A -85,B 0,C 180,E1 -24289.582,E2 -24289.582} C_VEL
LIN {X 0,Y 179.877,Z 403.056,A -85,B 0,C 180,E1 -24292.564,E2 -24292.564} C_VEL
LIN {X 0,Y 179.742,Z 402.891,A -85,B 0,C 180,E1 -24301.223,E2 -24301.223} C_VEL
LIN {X 0,Y 179.98,Z 403.329,A -85,B 0,C 180,E1 -24302.379,E2 -24302.379} C_VEL
LIN {X 0,Y 181.735,Z 406.947,A -85,B 0,C 180,E1 -24307.5,E2 -24307.5} C_VEL
LIN {X 0,Y 183.177,Z 408.409,A -85,B 0,C 180,E1 -24309.993,E2 -24309.993} C_VEL
LIN {X 0,Y 185.448,Z 412.075,A -85,B 0,C 180,E1 -24313.283,E2 -24313.283} C_VEL
LIN {X 0,Y 186.621,Z 413.6,A -85,B 0,C 180,E1 -24314.675,E2 -24314.675} C_VEL
LIN {X 0,Y 189.817,Z 418.261,A -85,B 0,C 180,E1 -24317.996,E2 -24317.996} C_VEL
LIN {X 0,Y 192.68,Z 422.513,A -85,B 0,C 180,E1 -24320.519,E2 -24320.519} C_VEL
LIN {X 0,Y 196.734,Z 428.947,A -85,B 0,C 180,E1 -24323.627,E2 -24323.627} C_VEL
LIN {X 0,Y 201.647,Z 437.418,A -85,B 0,C 180,E1 -24326.897,E2 -24326.897} C_VEL
LIN {X 0,Y 206.277,Z 446.404,A -85,B 0,C 180,E1 -24329.641,E2 -24329.641} C_VEL
LIN {X 0,Y 206.895,Z 447.906,A -85,B 0,C 180,E1 -24330.002,E2 -24330.002} C_VEL
LIN {X 0,Y 203.137,Z 491.802,A -85,B 0,C 180,E1 -24331.256,E2 -24331.256} C_VEL
LIN {X 0,Y 200.995,Z 505.499,A -85,B 0,C 180,E1 -24331.918,E2 -24331.918} C_VEL
LIN {X 0,Y 197.826,Z 519.585,A -85,B 0,C 180,E1 -24332.936,E2 -24332.936} C_VEL
LIN {X 0,Y 193.517,Z 533.606,A -85,B 0,C 180,E1 -24334.29,E2 -24334.29} C_VEL
LIN {X 0,Y 188.708,Z 546.112,A -85,B 0,C 180,E1 -24335.904,E2 -24335.904} C_VEL
LIN {X 0,Y 183.754,Z 557.001,A -85,B 0,C 180,E1 -24337.732,E2 -24337.732} C_VEL
LIN {X 0,Y 178.48,Z 566.988,A -85,B 0,C 180,E1 -24339.841,E2 -24339.841} C_VEL
LIN {X 0,Y 173.159,Z 575.898,A -85,B 0,C 180,E1 -24342.21,E2 -24342.21} C_VEL
LIN {X 0,Y 167.493,Z 584.629,A -85,B 0,C 180,E1 -24345.209,E2 -24345.209} C_VEL
LIN {X 0,Y 162.005,Z 592.275,A -85,B 0,C 180,E1 -24348.582,E2 -24348.582} C_VEL
LIN {X 0,Y 156.394,Z 599.342,A -85,B 0,C 180,E1 -24352.653,E2 -24352.653} C_VEL
LIN {X 0,Y 150.95,Z 605.659,A -85,B 0,C 180,E1 -24357.628,E2 -24357.628} C_VEL
LIN {X 0,Y 147.609,Z 609.26,A -85,B 0,C 180,E1 -24361.568,E2 -24361.568} C_VEL
LIN {X 0,Y 144.189,Z 612.758,A -85,B 0,C 180,E1 -24367.05,E2 -24367.05} C_VEL
LIN {X 0,Y 141.919,Z 614.839,A -85,B 0,C 180,E1 -24372.715,E2 -24372.715} C_VEL
LIN {X 0,Y 140.667,Z 615.571,A -85,B 0,C 180,E1 -24378.472,E2 -24378.472} C_VEL
LIN {X 0,Y 140.516,Z 614.971,A -85,B 0,C 180,E1 -24384.259,E2 -24384.259} C_VEL
LIN {X 0,Y 140.655,Z 613.878,A -85,B 0,C 180,E1 -24387.926,E2 -24387.926} C_VEL
LIN {X 0,Y 141.203,Z 611.585,A -85,B 0,C 180,E1 -24392.853,E2 -24392.853} C_VEL
LIN {X 0,Y 142.675,Z 607.577,A -85,B 0,C 180,E1 -24398.498,E2 -24398.498} C_VEL
LIN {X 0,Y 145.194,Z 602.035,A -85,B 0,C 180,E1 -24404.005,E2 -24404.005} C_VEL
LIN {X 0,Y 147.966,Z 596.772,A -85,B 0,C 180,E1 -24407.982,E2 -24407.982} C_VEL
LIN {X 0,Y 151.762,Z 589.216,A -85,B 0,C 180,E1 -24412.46,E2 -24412.46} C_VEL
LIN {X 0,Y 155.575,Z 581.351,A -85,B 0,C 180,E1 -24416.132,E2 -24416.132} C_VEL
LIN {X 0,Y 160.001,Z 571.863,A -85,B 0,C 180,E1 -24419.613,E2 -24419.613} C_VEL
LIN {X 0,Y 164.584,Z 561.344,A -85,B 0,C 180,E1 -24422.622,E2 -24422.622} C_VEL
LIN {X 0,Y 169.057,Z 549.72,A -85,B 0,C 180,E1 -24425.225,E2 -24425.225} C_VEL
LIN {X 0,Y 172.773,Z 538.381,A -85,B 0,C 180,E1 -24427.233,E2 -24427.233} C_VEL
LIN {X 0,Y 176.311,Z 526.082,A -85,B 0,C 180,E1 -24428.888,E2 -24428.888} C_VEL
LIN {X 0,Y 179.397,Z 512.464,A -85,B 0,C 180,E1 -24430.269,E2 -24430.269} C_VEL
LIN {X 0,Y 181.748,Z 498.192,A -85,B 0,C 180,E1 -24431.293,E2 -24431.293} C_VEL
LIN {X 0,Y 183.064,Z 485.208,A -85,B 0,C 180,E1 -24431.904,E2 -24431.904} C_VEL
LIN {X 0,Y 186.682,Z 430.222,A -85,B 0,C 180,E1 -24433.775,E2 -24433.775} C_VEL
LIN {X 0,Y 180.611,Z 418.011,A -85,B 0,C 180,E1 -24436.629,E2 -24436.629} C_VEL
LIN {X 0,Y 174.5,Z 407.517,A -85,B 0,C 180,E1 -24439.784,E2 -24439.784} C_VEL
LIN {X 0,Y 169.301,Z 399.641,A -85,B 0,C 180,E1 -24442.781,E2 -24442.781} C_VEL
LIN {X 0,Y 166.251,Z 395.253,A -85,B 0,C 180,E1 -24444.729,E2 -24444.729} C_VEL
LIN {X 0,Y 163.893,Z 391.952,A -85,B 0,C 180,E1 -24446.355,E2 -24446.355} C_VEL
LIN {X 0,Y 160.879,Z 387.84,A -85,B 0,C 180,E1 -24448.623,E2 -24448.623} C_VEL
LIN {X 0,Y 158.183,Z 384.365,A -85,B 0,C 180,E1 -24450.866,E2 -24450.866} C_VEL
LIN {X 0,Y 157.406,Z 383.211,A -85,B 0,C 180,E1 -24451.578,E2 -24451.578} C_VEL
LIN {X 0,Y 154.706,Z 380.492,A -85,B 0,C 180,E1 -24454.121,E2 -24454.121} C_VEL
LIN {X 0,Y 153.394,Z 377.981,A -85,B 0,C 180,E1 -24455.646,E2 -24455.646} C_VEL
LIN {X 0,Y 150.825,Z 376.274,A -85,B 0,C 180,E1 -24458.597,E2 -24458.597} C_VEL
LIN {X 0,Y 149.135,Z 373.451,A -85,B 0,C 180,E1 -24461.184,E2 -24461.184} C_VEL
LIN {X 0,Y 148.642,Z 372.269,A -85,B 0,C 180,E1 -24462.101,E2 -24462.101} C_VEL
LIN {X 0,Y 145.768,Z 370.636,A -85,B 0,C 180,E1 -24467.829,E2 -24467.829} C_VEL
LIN {X 0,Y 144.514,Z 368.915,A -85,B 0,C 180,E1 -24473.016,E2 -24473.016} C_VEL
LIN {X 0,Y 144.552,Z 367.826,A -85,B 0,C 180,E1 -24479.999,E2 -24479.999} C_VEL
LIN {X 0,Y 145.801,Z 370.57,A -85,B 0,C 180,E1 -24485.878,E2 -24485.878} C_VEL
LIN {X 0,Y 148.929,Z 372.485,A -85,B 0,C 180,E1 -24491.995,E2 -24491.995} C_VEL
LIN {X 0,Y 150.025,Z 375.068,A -85,B 0,C 180,E1 -24493.891,E2 -24493.891} C_VEL
LIN {X 0,Y 152.252,Z 377.394,A -85,B 0,C 180,E1 -24496.767,E2 -24496.767} C_VEL
LIN {X 0,Y 153.541,Z 378.249,A -85,B 0,C 180,E1 -24498.169,E2 -24498.169} C_VEL
LIN {X 0,Y 155.424,Z 381.414,A -85,B 0,C 180,E1 -24500.252,E2 -24500.252} C_VEL
LIN {X 0,Y 157.867,Z 383.746,A -85,B 0,C 180,E1 -24502.471,E2 -24502.471} C_VEL
LIN {X 0,Y 160.207,Z 387.143,A -85,B 0,C 180,E1 -24504.494,E2 -24504.494} C_VEL
LIN {X 0,Y 161.738,Z 388.836,A -85,B 0,C 180,E1 -24505.668,E2 -24505.668} C_VEL
LIN {X 0,Y 165.87,Z 394.569,A -85,B 0,C 180,E1 -24508.64,E2 -24508.64} C_VEL
LIN {X 0,Y 170.175,Z 400.724,A -85,B 0,C 180,E1 -24511.371,E2 -24511.371} C_VEL
LIN {X 0,Y 173.303,Z 405.946,A -85,B 0,C 180,E1 -24513.215,E2 -24513.215} C_VEL
LIN {X 0,Y 178.693,Z 417.063,A -85,B 0,C 180,E1 -24516.209,E2 -24516.209} C_VEL
LIN {X 0,Y 183.689,Z 429.13,A -85,B 0,C 180,E1 -24518.782,E2 -24518.782} C_VEL
LIN {X 0,Y 186.403,Z 436.83,A -85,B 0,C 180,E1 -24520.135,E2 -24520.135} C_VEL
LIN {X 0,Y 182.272,Z 495.979,A -85,B 0,C 180,E1 -24522.107,E2 -24522.107} C_VEL
LIN {X 0,Y 180.411,Z 510.662,A -85,B 0,C 180,E1 -24522.876,E2 -24522.876} C_VEL
LIN {X 0,Y 177.709,Z 524.749,A -85,B 0,C 180,E1 -24524.007,E2 -24524.007} C_VEL
LIN {X 0,Y 174.715,Z 536.426,A -85,B 0,C 180,E1 -24525.257,E2 -24525.257} C_VEL
LIN {X 0,Y 170.572,Z 549.754,A -85,B 0,C 180,E1 -24527.17,E2 -24527.17} C_VEL
LIN {X 0,Y 166.358,Z 561.615,A -85,B 0,C 180,E1 -24529.438,E2 -24529.438} C_VEL
LIN {X 0,Y 162.164,Z 571.759,A -85,B 0,C 180,E1 -24531.862,E2 -24531.862} C_VEL
LIN {X 0,Y 158.011,Z 581.103,A -85,B 0,C 180,E1 -24534.676,E2 -24534.676} C_VEL
LIN {X 0,Y 153.531,Z 590.448,A -85,B 0,C 180,E1 -24538.237,E2 -24538.237} C_VEL
LIN {X 0,Y 150.917,Z 595.838,A -85,B 0,C 180,E1 -24540.773,E2 -24540.773} C_VEL
LIN {X 0,Y 148.675,Z 599.174,A -85,B 0,C 180,E1 -24542.444,E2 -24542.444} C_VEL
LIN {X 0,Y 143.528,Z 604.153,A -85,B 0,C 180,E1 -24545.145,E2 -24545.145} C_VEL
LIN {X 0,Y 138.63,Z 608.587,A -85,B 0,C 180,E1 -24548.152,E2 -24548.152} C_VEL
LIN {X 0,Y 136.843,Z 611.01,A -85,B 0,C 180,E1 -24550.255,E2 -24550.255} C_VEL
LIN {X 0,Y 134.922,Z 615.316,A -85,B 0,C 180,E1 -24554.904,E2 -24554.904} C_VEL
LIN {X 0,Y 133.705,Z 619.389,A -85,B 0,C 180,E1 -24560.927,E2 -24560.927} C_VEL
LIN {X 0,Y 133.405,Z 621.985,A -85,B 0,C 180,E1 -24566.98,E2 -24566.98} C_VEL
LIN {X 0,Y 133.53,Z 622.759,A -85,B 0,C 180,E1 -24570,E2 -24570} C_VEL
LIN {X 0,Y 133.448,Z 623.269,A -85,B 0,C 180,E1 -24576.046,E2 -24576.046} C_VEL
LIN {X 0,Y 134.266,Z 622.455,A -85,B 0,C 180,E1 -24582.085,E2 -24582.085} C_VEL
LIN {X 0,Y 136.24,Z 620.313,A -85,B 0,C 180,E1 -24588.029,E2 -24588.029} C_VEL
LIN {X 0,Y 139.621,Z 616.797,A -85,B 0,C 180,E1 -24593.746,E2 -24593.746} C_VEL
LIN {X 0,Y 144.146,Z 611.802,A -85,B 0,C 180,E1 -24599.179,E2 -24599.179} C_VEL
LIN {X 0,Y 150,Z 605.19,A -85,B 0,C 180,E1 -24604.21,E2 -24604.21} C_VEL
LIN {X 0,Y 155.978,Z 597.858,A -85,B 0,C 180,E1 -24608.282,E2 -24608.282} C_VEL
LIN {X 0,Y 162.838,Z 588.772,A -85,B 0,C 180,E1 -24611.986,E2 -24611.986} C_VEL
LIN {X 0,Y 169.098,Z 579.286,A -85,B 0,C 180,E1 -24614.953,E2 -24614.953} C_VEL
LIN {X 0,Y 175.231,Z 568.797,A -85,B 0,C 180,E1 -24617.472,E2 -24617.472} C_VEL
LIN {X 0,Y 181.135,Z 557.233,A -85,B 0,C 180,E1 -24619.59,E2 -24619.59} C_VEL
LIN {X 0,Y 186.753,Z 544.4,A -85,B 0,C 180,E1 -24621.339,E2 -24621.339} C_VEL
LIN {X 0,Y 191.227,Z 531.855,A -85,B 0,C 180,E1 -24622.631,E2 -24622.631} C_VEL
LIN {X 0,Y 195.117,Z 517.901,A -85,B 0,C 180,E1 -24623.697,E2 -24623.697} C_VEL
LIN {X 0,Y 197.879,Z 504.114,A -85,B 0,C 180,E1 -24624.438,E2 -24624.438} C_VEL
LIN {X 0,Y 199.729,Z 488.996,A -85,B 0,C 180,E1 -24624.944,E2 -24624.944} C_VEL
LIN {X 0,Y 202.397,Z 456.463,A -85,B 0,C 180,E1 -24625.879,E2 -24625.879} C_VEL
LIN {X 0,Y 198.795,Z 447.222,A -85,B 0,C 180,E1 -24628.282,E2 -24628.282} C_VEL
LIN {X 0,Y 195.193,Z 438.803,A -85,B 0,C 180,E1 -24630.919,E2 -24630.919} C_VEL
LIN {X 0,Y 191.478,Z 430.995,A -85,B 0,C 180,E1 -24633.963,E2 -24633.963} C_VEL
LIN {X 0,Y 188.436,Z 425.296,A -85,B 0,C 180,E1 -24636.807,E2 -24636.807} C_VEL
LIN {X 0,Y 187.003,Z 423.136,A -85,B 0,C 180,E1 -24638.262,E2 -24638.262} C_VEL
LIN {X 0,Y 184.548,Z 419.394,A -85,B 0,C 180,E1 -24641.114,E2 -24641.114} C_VEL
LIN {X 0,Y 182.186,Z 415.988,A -85,B 0,C 180,E1 -24644.492,E2 -24644.492} C_VEL
LIN {X 0,Y 181.66,Z 414.989,A -85,B 0,C 180,E1 -24645.435,E2 -24645.435} C_VEL
LIN {X 0,Y 179.412,Z 412.054,A -85,B 0,C 180,E1 -24650.503,E2 -24650.503} C_VEL
LIN {X 0,Y 178.857,Z 410.039,A -85,B 0,C 180,E1 -24653.231,E2 -24653.231} C_VEL
LIN {X 0,Y 178.874,Z 409.938,A -85,B 0,C 180,E1 -24661.229,E2 -24661.229} C_VEL
LIN {X 0,Y 179.113,Z 410.71,A -85,B 0,C 180,E1 -24662.531,E2 -24662.531} C_VEL
LIN {X 0,Y 181.041,Z 414.287,A -85,B 0,C 180,E1 -24667.88,E2 -24667.88} C_VEL
LIN {X 0,Y 181.968,Z 415.322,A -85,B 0,C 180,E1 -24669.517,E2 -24669.517} C_VEL
LIN {X 0,Y 184.201,Z 418.945,A -85,B 0,C 180,E1 -24672.884,E2 -24672.884} C_VEL
LIN {X 0,Y 185.23,Z 420.468,A -85,B 0,C 180,E1 -24674.173,E2 -24674.173} C_VEL
LIN {X 0,Y 188.186,Z 424.911,A -85,B 0,C 180,E1 -24677.384,E2 -24677.384} C_VEL
LIN {X 0,Y 190.99,Z 429.29,A -85,B 0,C 180,E1 -24679.971,E2 -24679.971} C_VEL
LIN {X 0,Y 194.711,Z 435.451,A -85,B 0,C 180,E1 -24682.955,E2 -24682.955} C_VEL
LIN {X 0,Y 199.276,Z 443.658,A -85,B 0,C 180,E1 -24686.143,E2 -24686.143} C_VEL
LIN {X 0,Y 202.813,Z 450.718,A -85,B 0,C 180,E1 -24688.368,E2 -24688.368} C_VEL
LIN {X 0,Y 199.237,Z 491.931,A -85,B 0,C 180,E1 -24689.577,E2 -24689.577} C_VEL
LIN {X 0,Y 197.089,Z 505.332,A -85,B 0,C 180,E1 -24690.211,E2 -24690.211} C_VEL
LIN {X 0,Y 194.018,Z 518.769,A -85,B 0,C 180,E1 -24691.157,E2 -24691.157} C_VEL
LIN {X 0,Y 190.197,Z 531.229,A -85,B 0,C 180,E1 -24692.303,E2 -24692.303} C_VEL
LIN {X 0,Y 185.222,Z 544.237,A -85,B 0,C 180,E1 -24693.902,E2 -24693.902} C_VEL
LIN {X 0,Y 179.987,Z 555.667,A -85,B 0,C 180,E1 -24695.747,E2 -24695.747} C_VEL
LIN {X 0,Y 175.141,Z 564.787,A -85,B 0,C 180,E1 -24697.58,E2 -24697.58} C_VEL
LIN {X 0,Y 169.456,Z 574.094,A -85,B 0,C 180,E1 -24699.893,E2 -24699.893} C_VEL
LIN {X 0,Y 163.273,Z 583.387,A -85,B 0,C 180,E1 -24702.968,E2 -24702.968} C_VEL
LIN {X 0,Y 157.575,Z 591.106,A -85,B 0,C 180,E1 -24706.267,E2 -24706.267} C_VEL
LIN {X 0,Y 152.35,Z 597.497,A -85,B 0,C 180,E1 -24709.773,E2 -24709.773} C_VEL
LIN {X 0,Y 147.649,Z 602.74,A -85,B 0,C 180,E1 -24713.489,E2 -24713.489} C_VEL
LIN {X 0,Y 142.435,Z 608.25,A -85,B 0,C 180,E1 -24718.797,E2 -24718.797} C_VEL
LIN {X 0,Y 139.277,Z 611.295,A -85,B 0,C 180,E1 -24722.991,E2 -24722.991} C_VEL
LIN {X 0,Y 136.177,Z 614.111,A -85,B 0,C 180,E1 -24728.823,E2 -24728.823} C_VEL
LIN {X 0,Y 134.166,Z 615.549,A -85,B 0,C 180,E1 -24734.817,E2 -24734.817} C_VEL
LIN {X 0,Y 133.411,Z 615.648,A -85,B 0,C 180,E1 -24740.907,E2 -24740.907} C_VEL
LIN {X 0,Y 133.411,Z 615.201,A -85,B 0,C 180,E1 -24743.952,E2 -24743.952} C_VEL
LIN {X 0,Y 133.58,Z 613.882,A -85,B 0,C 180,E1 -24748.518,E2 -24748.518} C_VEL
LIN {X 0,Y 134.119,Z 611.883,A -85,B 0,C 180,E1 -24753.004,E2 -24753.004} C_VEL
LIN {X 0,Y 135.683,Z 607.917,A -85,B 0,C 180,E1 -24758.939,E2 -24758.939} C_VEL
LIN {X 0,Y 138.331,Z 602.418,A -85,B 0,C 180,E1 -24764.716,E2 -24764.716} C_VEL
LIN {X 0,Y 142.037,Z 595.651,A -85,B 0,C 180,E1 -24769.925,E2 -24769.925} C_VEL
LIN {X 0,Y 145.853,Z 588.475,A -85,B 0,C 180,E1 -24774.177,E2 -24774.177} C_VEL
LIN {X 0,Y 150.025,Z 580.409,A -85,B 0,C 180,E1 -24777.933,E2 -24777.933} C_VEL
LIN {X 0,Y 154.78,Z 570.688,A -85,B 0,C 180,E1 -24781.477,E2 -24781.477} C_VEL
LIN {X 0,Y 159.589,Z 559.898,A -85,B 0,C 180,E1 -24784.54,E2 -24784.54} C_VEL
LIN {X 0,Y 164.336,Z 547.927,A -85,B 0,C 180,E1 -24787.161,E2 -24787.161} C_VEL
LIN {X 0,Y 168.213,Z 536.145,A -85,B 0,C 180,E1 -24789.191,E2 -24789.191} C_VEL
LIN {X 0,Y 171.936,Z 523.195,A -85,B 0,C 180,E1 -24790.843,E2 -24790.843} C_VEL
LIN {X 0,Y 175.015,Z 509.09,A -85,B 0,C 180,E1 -24792.171,E2 -24792.171} C_VEL
LIN {X 0,Y 177.19,Z 494.518,A -85,B 0,C 180,E1 -24793.13,E2 -24793.13} C_VEL
LIN {X 0,Y 178.851,Z 475.14,A -85,B 0,C 180,E1 -24793.878,E2 -24793.878} C_VEL
LIN {X 0,Y 181.736,Z 432.851,A -85,B 0,C 180,E1 -24795.328,E2 -24795.328} C_VEL
LIN {X 0,Y 176.423,Z 421.971,A -85,B 0,C 180,E1 -24798.024,E2 -24798.024} C_VEL
LIN {X 0,Y 171.075,Z 412.611,A -85,B 0,C 180,E1 -24800.981,E2 -24800.981} C_VEL
LIN {X 0,Y 166.231,Z 405.069,A -85,B 0,C 180,E1 -24803.962,E2 -24803.962} C_VEL
LIN {X 0,Y 161.819,Z 398.451,A -85,B 0,C 180,E1 -24807.057,E2 -24807.057} C_VEL
LIN {X 0,Y 158.388,Z 393.794,A -85,B 0,C 180,E1 -24809.772,E2 -24809.772} C_VEL
LIN {X 0,Y 155.778,Z 390.091,A -85,B 0,C 180,E1 -24812.127,E2 -24812.127} C_VEL
LIN {X 0,Y 152.6,Z 386.48,A -85,B 0,C 180,E1 -24815.332,E2 -24815.332} C_VEL
LIN {X 0,Y 151.767,Z 384.8,A -85,B 0,C 180,E1 -24816.372,E2 -24816.372} C_VEL
LIN {X 0,Y 149.032,Z 382.575,A -85,B 0,C 180,E1 -24819.781,E2 -24819.781} C_VEL
LIN {X 0,Y 147.461,Z 379.456,A -85,B 0,C 180,E1 -24822.504,E2 -24822.504} C_VEL
LIN {X 0,Y 143.561,Z 375.843,A -85,B 0,C 180,E1 -24833.675,E2 -24833.675} C_VEL
LIN {X 0,Y 143.435,Z 375.134,A -85,B 0,C 180,E1 -24837.191,E2 -24837.191} C_VEL
LIN {X 0,Y 143.685,Z 375.276,A -85,B 0,C 180,E1 -24840.349,E2 -24840.349} C_VEL
LIN {X 0,Y 145.331,Z 377.982,A -85,B 0,C 180,E1 -24846.943,E2 -24846.943} C_VEL
LIN {X 0,Y 147.514,Z 379.372,A -85,B 0,C 180,E1 -24851.203,E2 -24851.203} C_VEL
LIN {X 0,Y 148.912,Z 382.227,A -85,B 0,C 180,E1 -24853.648,E2 -24853.648} C_VEL
LIN {X 0,Y 151.373,Z 384.535,A -85,B 0,C 180,E1 -24856.824,E2 -24856.824} C_VEL
LIN {X 0,Y 151.955,Z 385.251,A -85,B 0,C 180,E1 -24857.516,E2 -24857.516} C_VEL
LIN {X 0,Y 154.257,Z 388.635,A -85,B 0,C 180,E1 -24860.079,E2 -24860.079} C_VEL
LIN {X 0,Y 155.942,Z 390.372,A -85,B 0,C 180,E1 -24861.674,E2 -24861.674} C_VEL
LIN {X 0,Y 158.636,Z 394.048,A -85,B 0,C 180,E1 -24864.066,E2 -24864.066} C_VEL
LIN {X 0,Y 162.865,Z 399.921,A -85,B 0,C 180,E1 -24867.344,E2 -24867.344} C_VEL
LIN {X 0,Y 167.464,Z 406.774,A -85,B 0,C 180,E1 -24870.456,E2 -24870.456} C_VEL
LIN {X 0,Y 170.351,Z 411.802,A -85,B 0,C 180,E1 -24872.258,E2 -24872.258} C_VEL
LIN {X 0,Y 175.57,Z 423.195,A -85,B 0,C 180,E1 -24875.341,E2 -24875.341} C_VEL
LIN {X 0,Y 179.906,Z 434.41,A -85,B 0,C 180,E1 -24877.733,E2 -24877.733} C_VEL
LIN {X 0,Y 181.474,Z 439.06,A -85,B 0,C 180,E1 -24878.577,E2 -24878.577} C_VEL
LIN {X 0,Y 177.24,Z 496.71,A -85,B 0,C 180,E1 -24880.514,E2 -24880.514} C_VEL
LIN {X 0,Y 175.352,Z 510.839,A -85,B 0,C 180,E1 -24881.283,E2 -24881.283} C_VEL
LIN {X 0,Y 172.552,Z 524.796,A -85,B 0,C 180,E1 -24882.421,E2 -24882.421} C_VEL
LIN {X 0,Y 169.185,Z 537.342,A -85,B 0,C 180,E1 -24883.802,E2 -24883.802} C_VEL
LIN {X 0,Y 164.878,Z 550.428,A -85,B 0,C 180,E1 -24885.736,E2 -24885.736} C_VEL
LIN {X 0,Y 160.433,Z 562.31,A -85,B 0,C 180,E1 -24888.087,E2 -24888.087} C_VEL
LIN {X 0,Y 155.683,Z 573.143,A -85,B 0,C 180,E1 -24890.803,E2 -24890.803} C_VEL
LIN {X 0,Y 151.398,Z 582.228,A -85,B 0,C 180,E1 -24893.712,E2 -24893.712} C_VEL
LIN {X 0,Y 146.751,Z 591.349,A -85,B 0,C 180,E1 -24897.401,E2 -24897.401} C_VEL
LIN {X 0,Y 142.239,Z 600.073,A -85,B 0,C 180,E1 -24902.006,E2 -24902.006} C_VEL
LIN {X 0,Y 139.153,Z 606.195,A -85,B 0,C 180,E1 -24906.169,E2 -24906.169} C_VEL
LIN {X 0,Y 136.843,Z 611.01,A -85,B 0,C 180,E1 -24910.255,E2 -24910.255} C_VEL
LIN {X 0,Y 135.197,Z 613.271,A -85,B 0,C 180,E1 -24912.445,E2 -24912.445} C_VEL
LIN {X 0,Y 131.064,Z 616.365,A -85,B 0,C 180,E1 -24916.089,E2 -24916.089} C_VEL
LIN {X 0,Y 127.939,Z 618.409,A -85,B 0,C 180,E1 -24919.213,E2 -24919.213} C_VEL
LIN {X 0,Y 126.577,Z 619.745,A -85,B 0,C 180,E1 -24921.747,E2 -24921.747} C_VEL
LIN {X 0,Y 126.431,Z 620.134,A -85,B 0,C 180,E1 -24922.621,E2 -24922.621} C_VEL
LIN {X 0,Y 126.306,Z 621.74,A -85,B 0,C 180,E1 -24926.81,E2 -24926.81} C_VEL
LIN {X 0,Y 126.426,Z 622.533,A -85,B 0,C 180,E1 -24930,E2 -24930} C_VEL
LIN {X 0,Y 126.388,Z 623.075,A -85,B 0,C 180,E1 -24936.385,E2 -24936.385} C_VEL
LIN {X 0,Y 127.304,Z 622.291,A -85,B 0,C 180,E1 -24942.757,E2 -24942.757} C_VEL
LIN {X 0,Y 129.478,Z 620.181,A -85,B 0,C 180,E1 -24949.006,E2 -24949.006} C_VEL
LIN {X 0,Y 133.12,Z 616.699,A -85,B 0,C 180,E1 -24954.983,E2 -24954.983} C_VEL
LIN {X 0,Y 137.962,Z 611.74,A -85,B 0,C 180,E1 -24960.624,E2 -24960.624} C_VEL
LIN {X 0,Y 144.153,Z 605.166,A -85,B 0,C 180,E1 -24965.805,E2 -24965.805} C_VEL
LIN {X 0,Y 150.461,Z 597.875,A -85,B 0,C 180,E1 -24969.959,E2 -24969.959} C_VEL
LIN {X 0,Y 157.632,Z 588.862,A -85,B 0,C 180,E1 -24973.713,E2 -24973.713} C_VEL
LIN {X 0,Y 164.642,Z 578.636,A -85,B 0,C 180,E1 -24976.924,E2 -24976.924} C_VEL
LIN {X 0,Y 171.133,Z 567.949,A -85,B 0,C 180,E1 -24979.44,E2 -24979.44} C_VEL
LIN {X 0,Y 177.26,Z 556.251,A -85,B 0,C 180,E1 -24981.538,E2 -24981.538} C_VEL
LIN {X 0,Y 182.41,Z 544.82,A -85,B 0,C 180,E1 -24983.077,E2 -24983.077} C_VEL
LIN {X 0,Y 187.019,Z 532.434,A -85,B 0,C 180,E1 -24984.353,E2 -24984.353} C_VEL
LIN {X 0,Y 191.006,Z 518.765,A -85,B 0,C 180,E1 -24985.402,E2 -24985.402} C_VEL
LIN {X 0,Y 194.021,Z 504.5,A -85,B 0,C 180,E1 -24986.173,E2 -24986.173} C_VEL
LIN {X 0,Y 195.963,Z 489.64,A -85,B 0,C 180,E1 -24986.674,E2 -24986.674} C_VEL
LIN {X 0,Y 198.531,Z 459.275,A -85,B 0,C 180,E1 -24987.548,E2 -24987.548} C_VEL
LIN {X 0,Y 194.574,Z 448.902,A -85,B 0,C 180,E1 -24990.467,E2 -24990.467} C_VEL
LIN {X 0,Y 190.803,Z 440.127,A -85,B 0,C 180,E1 -24993.585,E2 -24993.585} C_VEL
LIN {X 0,Y 187.396,Z 433.049,A -85,B 0,C 180,E1 -24996.824,E2 -24996.824} C_VEL
LIN {X 0,Y 185.515,Z 429.841,A -85,B 0,C 180,E1 -24998.821,E2 -24998.821} C_VEL
LIN {X 0,Y 183.108,Z 426.066,A -85,B 0,C 180,E1 -25001.758,E2 -25001.758} C_VEL
LIN {X 0,Y 180.827,Z 422.511,A -85,B 0,C 180,E1 -25005.266,E2 -25005.266} C_VEL
LIN {X 0,Y 180.287,Z 421.689,A -85,B 0,C 180,E1 -25006.271,E2 -25006.271} C_VEL
LIN {X 0,Y 178.368,Z 418.855,A -85,B 0,C 180,E1 -25011.076,E2 -25011.076} C_VEL
LIN {X 0,Y 177.986,Z 417.162,A -85,B 0,C 180,E1 -25013.198,E2 -25013.198} C_VEL
LIN {X 0,Y 177.8,Z 416.798,A -85,B 0,C 180,E1 -25020.001,E2 -25020.001} C_VEL
LIN {X 0,Y 178.082,Z 417.354,A -85,B 0,C 180,E1 -25021.748,E2 -25021.748} C_VEL
LIN {X 0,Y 179.852,Z 421.102,A -85,B 0,C 180,E1 -25027.297,E2 -25027.297} C_VEL
LIN {X 0,Y 180.734,Z 422.09,A -85,B 0,C 180,E1 -25028.949,E2 -25028.949} C_VEL
LIN {X 0,Y 182.937,Z 425.788,A -85,B 0,C 180,E1 -25032.446,E2 -25032.446} C_VEL
LIN {X 0,Y 184.077,Z 427.708,A -85,B 0,C 180,E1 -25033.947,E2 -25033.947} C_VEL
LIN {X 0,Y 186.411,Z 431.262,A -85,B 0,C 180,E1 -25036.584,E2 -25036.584} C_VEL
LIN {X 0,Y 189.248,Z 435.956,A -85,B 0,C 180,E1 -25039.35,E2 -25039.35} C_VEL
LIN {X 0,Y 192.676,Z 441.891,A -85,B 0,C 180,E1 -25042.238,E2 -25042.238} C_VEL
LIN {X 0,Y 196.494,Z 449.053,A -85,B 0,C 180,E1 -25045.064,E2 -25045.064} C_VEL
LIN {X 0,Y 198.954,Z 454.133,A -85,B 0,C 180,E1 -25046.735,E2 -25046.735} C_VEL
LIN {X 0,Y 195.382,Z 492.806,A -85,B 0,C 180,E1 -25047.848,E2 -25047.848} C_VEL
LIN {X 0,Y 193.093,Z 506.404,A -85,B 0,C 180,E1 -25048.508,E2 -25048.508} C_VEL
LIN {X 0,Y 189.751,Z 520.238,A -85,B 0,C 180,E1 -25049.498,E2 -25049.498} C_VEL
LIN {X 0,Y 185.16,Z 534.202,A -85,B 0,C 180,E1 -25050.825,E2 -25050.825} C_VEL
LIN {X 0,Y 180.025,Z 546.671,A -85,B 0,C 180,E1 -25052.414,E2 -25052.414} C_VEL
LIN {X 0,Y 174.318,Z 558.283,A -85,B 0,C 180,E1 -25054.365,E2 -25054.365} C_VEL
LIN {X 0,Y 168.443,Z 568.48,A -85,B 0,C 180,E1 -25056.568,E2 -25056.568} C_VEL
LIN {X 0,Y 162.709,Z 577.208,A -85,B 0,C 180,E1 -25058.971,E2 -25058.971} C_VEL
LIN {X 0,Y 156.163,Z 586.272,A -85,B 0,C 180,E1 -25062.237,E2 -25062.237} C_VEL
LIN {X 0,Y 149.594,Z 594.42,A -85,B 0,C 180,E1 -25066.137,E2 -25066.137} C_VEL
LIN {X 0,Y 143.515,Z 601.143,A -85,B 0,C 180,E1 -25070.461,E2 -25070.461} C_VEL
LIN {X 0,Y 137.59,Z 607.074,A -85,B 0,C 180,E1 -25075.816,E2 -25075.816} C_VEL
LIN {X 0,Y 132.872,Z 611.399,A -85,B 0,C 180,E1 -25081.574,E2 -25081.574} C_VEL
LIN {X 0,Y 129.47,Z 614.252,A -85,B 0,C 180,E1 -25087.668,E2 -25087.668} C_VEL
LIN {X 0,Y 127.251,Z 615.726,A -85,B 0,C 180,E1 -25093.97,E2 -25093.97} C_VEL
LIN {X 0,Y 126.334,Z 615.861,A -85,B 0,C 180,E1 -25100.393,E2 -25100.393} C_VEL
LIN {X 0,Y 126.294,Z 615.432,A -85,B 0,C 180,E1 -25103.61,E2 -25103.61} C_VEL
LIN {X 0,Y 126.528,Z 613.96,A -85,B 0,C 180,E1 -25108.961,E2 -25108.961} C_VEL
LIN {X 0,Y 127.039,Z 612.174,A -85,B 0,C 180,E1 -25113.171,E2 -25113.171} C_VEL
LIN {X 0,Y 128.684,Z 608.257,A -85,B 0,C 180,E1 -25119.43,E2 -25119.43} C_VEL
LIN {X 0,Y 131.487,Z 602.799,A -85,B 0,C 180,E1 -25125.5,E2 -25125.5} C_VEL
LIN {X 0,Y 135.051,Z 596.719,A -85,B 0,C 180,E1 -25130.49,E2 -25130.49} C_VEL
LIN {X 0,Y 139.429,Z 588.949,A -85,B 0,C 180,E1 -25135.368,E2 -25135.368} C_VEL
LIN {X 0,Y 143.818,Z 580.939,A -85,B 0,C 180,E1 -25139.253,E2 -25139.253} C_VEL
LIN {X 0,Y 148.791,Z 571.285,A -85,B 0,C 180,E1 -25142.9,E2 -25142.9} C_VEL
LIN {X 0,Y 153.828,Z 560.572,A -85,B 0,C 180,E1 -25146.03,E2 -25146.03} C_VEL
LIN {X 0,Y 158.773,Z 548.699,A -85,B 0,C 180,E1 -25148.698,E2 -25148.698} C_VEL
LIN {X 0,Y 162.807,Z 537.046,A -85,B 0,C 180,E1 -25150.76,E2 -25150.76} C_VEL
LIN {X 0,Y 166.952,Z 523.276,A -85,B 0,C 180,E1 -25152.543,E2 -25152.543} C_VEL
LIN {X 0,Y 170.136,Z 509.127,A -85,B 0,C 180,E1 -25153.882,E2 -25153.882} C_VEL
LIN {X 0,Y 172.307,Z 495.294,A -85,B 0,C 180,E1 -25154.801,E2 -25154.801} C_VEL
LIN {X 0,Y 173.921,Z 477.871,A -85,B 0,C 180,E1 -25155.497,E2 -25155.497} C_VEL
LIN {X 0,Y 176.927,Z 435.528,A -85,B 0,C 180,E1 -25156.966,E2 -25156.966} C_VEL
LIN {X 0,Y 172.076,Z 425.537,A -85,B 0,C 180,E1 -25159.631,E2 -25159.631} C_VEL
LIN {X 0,Y 167.476,Z 417.329,A -85,B 0,C 180,E1 -25162.378,E2 -25162.378} C_VEL
LIN {X 0,Y 163.392,Z 410.743,A -85,B 0,C 180,E1 -25165.076,E2 -25165.076} C_VEL
LIN {X 0,Y 159.599,Z 404.731,A -85,B 0,C 180,E1 -25167.908,E2 -25167.908} C_VEL
LIN {X 0,Y 156.114,Z 399.957,A -85,B 0,C 180,E1 -25170.82,E2 -25170.82} C_VEL
LIN {X 0,Y 153.433,Z 396.068,A -85,B 0,C 180,E1 -25173.413,E2 -25173.413} C_VEL
LIN {X 0,Y 150.869,Z 392.996,A -85,B 0,C 180,E1 -25176.192,E2 -25176.192} C_VEL
LIN {X 0,Y 150.087,Z 391.481,A -85,B 0,C 180,E1 -25177.216,E2 -25177.216} C_VEL
LIN {X 0,Y 147.388,Z 388.955,A -85,B 0,C 180,E1 -25180.862,E2 -25180.862} C_VEL
LIN {X 0,Y 145.946,Z 386.073,A -85,B 0,C 180,E1 -25183.586,E2 -25183.586} C_VEL
LIN {X 0,Y 142.625,Z 382.776,A -85,B 0,C 180,E1 -25194.343,E2 -25194.343} C_VEL
LIN {X 0,Y 142.567,Z 382.194,A -85,B 0,C 180,E1 -25197.173,E2 -25197.173} C_VEL
LIN {X 0,Y 142.788,Z 382.397,A -85,B 0,C 180,E1 -25200.219,E2 -25200.219} C_VEL
LIN {X 0,Y 144.466,Z 385.064,A -85,B 0,C 180,E1 -25206.985,E2 -25206.985} C_VEL
LIN {X 0,Y 146.162,Z 386.189,A -85,B 0,C 180,E1 -25210.436,E2 -25210.436} C_VEL
LIN {X 0,Y 147.701,Z 389.192,A -85,B 0,C 180,E1 -25213.237,E2 -25213.237} C_VEL
LIN {X 0,Y 150.238,Z 391.789,A -85,B 0,C 180,E1 -25216.627,E2 -25216.627} C_VEL
LIN {X 0,Y 152.683,Z 395.382,A -85,B 0,C 180,E1 -25219.482,E2 -25219.482} C_VEL
LIN {X 0,Y 153.993,Z 396.856,A -85,B 0,C 180,E1 -25220.795,E2 -25220.795} C_VEL
LIN {X 0,Y 157.615,Z 401.959,A -85,B 0,C 180,E1 -25224.117,E2 -25224.117} C_VEL
LIN {X 0,Y 161.271,Z 407.303,A -85,B 0,C 180,E1 -25227.014,E2 -25227.014} C_VEL
LIN {X 0,Y 166.156,Z 415.097,A -85,B 0,C 180,E1 -25230.413,E2 -25230.413} C_VEL
LIN {X 0,Y 170.882,Z 425.527,A -85,B 0,C 180,E1 -25233.471,E2 -25233.471} C_VEL
LIN {X 0,Y 175.178,Z 436.652,A -85,B 0,C 180,E1 -25236.046,E2 -25236.046} C_VEL
LIN {X 0,Y 176.688,Z 441.252,A -85,B 0,C 180,E1 -25236.932,E2 -25236.932} C_VEL
LIN {X 0,Y 172.417,Z 496.946,A -85,B 0,C 180,E1 -25238.819,E2 -25238.819} C_VEL
LIN {X 0,Y 170.291,Z 511.759,A -85,B 0,C 180,E1 -25239.652,E2 -25239.652} C_VEL
LIN {X 0,Y 167.224,Z 525.971,A -85,B 0,C 180,E1 -25240.846,E2 -25240.846} C_VEL
LIN {X 0,Y 163.761,Z 538.22,A -85,B 0,C 180,E1 -25242.245,E2 -25242.245} C_VEL
LIN {X 0,Y 159.293,Z 551.098,A -85,B 0,C 180,E1 -25244.199,E2 -25244.199} C_VEL
LIN {X 0,Y 154.997,Z 562.088,A -85,B 0,C 180,E1 -25246.425,E2 -25246.425} C_VEL
LIN {X 0,Y 150.231,Z 572.556,A -85,B 0,C 180,E1 -25249.086,E2 -25249.086} C_VEL
LIN {X 0,Y 144.818,Z 583.345,A -85,B 0,C 180,E1 -25252.656,E2 -25252.656} C_VEL
LIN {X 0,Y 140.012,Z 592.246,A -85,B 0,C 180,E1 -25256.486,E2 -25256.486} C_VEL
LIN {X 0,Y 135.949,Z 599.649,A -85,B 0,C 180,E1 -25260.587,E2 -25260.587} C_VEL
LIN {X 0,Y 132.609,Z 605.813,A -85,B 0,C 180,E1 -25264.914,E2 -25264.914} C_VEL
LIN {X 0,Y 129.284,Z 612.358,A -85,B 0,C 180,E1 -25270.964,E2 -25270.964} C_VEL
LIN {X 0,Y 127.221,Z 617.236,A -85,B 0,C 180,E1 -25277.234,E2 -25277.234} C_VEL
LIN {X 0,Y 126.431,Z 620.134,A -85,B 0,C 180,E1 -25282.621,E2 -25282.621} C_VEL
LIN {X 0,Y 126.025,Z 620.895,A -85,B 0,C 180,E1 -25284.366,E2 -25284.366} C_VEL
LIN {X 0,Y 124.593,Z 621.807,A -85,B 0,C 180,E1 -25286.966,E2 -25286.966} C_VEL
LIN {X 0,Y 121.395,Z 622.717,A -85,B 0,C 180,E1 -25291.366,E2 -25291.366} C_VEL
LIN {X 0,Y 119.539,Z 622.928,A -85,B 0,C 180,E1 -25295.095,E2 -25295.095} C_VEL
LIN {X 0,Y 119.315,Z 622.864,A -85,B 0,C 180,E1 -25297.019,E2 -25297.019} C_VEL
LIN {X 0,Y 120.351,Z 622.128,A -85,B 0,C 180,E1 -25303.508,E2 -25303.508} C_VEL
LIN {X 0,Y 122.762,Z 620.05,A -85,B 0,C 180,E1 -25310.089,E2 -25310.089} C_VEL
LIN {X 0,Y 126.684,Z 616.601,A -85,B 0,C 180,E1 -25316.347,E2 -25316.347} C_VEL
LIN {X 0,Y 131.869,Z 611.678,A -85,B 0,C 180,E1 -25322.204,E2 -25322.204} C_VEL
LIN {X 0,Y 138.42,Z 605.142,A -85,B 0,C 180,E1 -25327.536,E2 -25327.536} C_VEL
LIN {X 0,Y 145.063,Z 597.893,A -85,B 0,C 180,E1 -25331.77,E2 -25331.77} C_VEL
LIN {X 0,Y 152.579,Z 588.948,A -85,B 0,C 180,E1 -25335.556,E2 -25335.556} C_VEL
LIN {X 0,Y 159.465,Z 579.404,A -85,B 0,C 180,E1 -25338.618,E2 -25338.618} C_VEL
LIN {X 0,Y 165.974,Z 569.237,A -85,B 0,C 180,E1 -25341.082,E2 -25341.082} C_VEL
LIN {X 0,Y 172.286,Z 557.848,A -85,B 0,C 180,E1 -25343.181,E2 -25343.181} C_VEL
LIN {X 0,Y 178.251,Z 545.245,A -85,B 0,C 180,E1 -25344.895,E2 -25344.895} C_VEL
LIN {X 0,Y 182.996,Z 533.021,A -85,B 0,C 180,E1 -25346.149,E2 -25346.149} C_VEL
LIN {X 0,Y 187.076,Z 519.653,A -85,B 0,C 180,E1 -25347.177,E2 -25347.177} C_VEL
LIN {X 0,Y 190.297,Z 505.179,A -85,B 0,C 180,E1 -25347.963,E2 -25347.963} C_VEL
LIN {X 0,Y 192.311,Z 490.981,A -85,B 0,C 180,E1 -25348.448,E2 -25348.448} C_VEL
LIN {X 0,Y 194.831,Z 462.127,A -85,B 0,C 180,E1 -25349.285,E2 -25349.285} C_VEL
LIN {X 0,Y 191.151,Z 452.308,A -85,B 0,C 180,E1 -25352.269,E2 -25352.269} C_VEL
LIN {X 0,Y 187.657,Z 443.866,A -85,B 0,C 180,E1 -25355.493,E2 -25355.493} C_VEL
LIN {X 0,Y 184.841,Z 437.921,A -85,B 0,C 180,E1 -25358.477,E2 -25358.477} C_VEL
LIN {X 0,Y 181.695,Z 432.706,A -85,B 0,C 180,E1 -25362.412,E2 -25362.412} C_VEL
LIN {X 0,Y 179.538,Z 429.128,A -85,B 0,C 180,E1 -25365.974,E2 -25365.974} C_VEL
LIN {X 0,Y 177.22,Z 425.198,A -85,B 0,C 180,E1 -25372.279,E2 -25372.279} C_VEL
LIN {X 0,Y 177.053,Z 424.187,A -85,B 0,C 180,E1 -25373.52,E2 -25373.52} C_VEL
LIN {X 0,Y 177.078,Z 424,A -85,B 0,C 180,E1 -25380.931,E2 -25380.931} C_VEL
LIN {X 0,Y 178.846,Z 428.092,A -85,B 0,C 180,E1 -25387.055,E2 -25387.055} C_VEL
LIN {X 0,Y 179.561,Z 429.017,A -85,B 0,C 180,E1 -25388.476,E2 -25388.476} C_VEL
LIN {X 0,Y 182.221,Z 433.578,A -85,B 0,C 180,E1 -25392.761,E2 -25392.761} C_VEL
LIN {X 0,Y 184.933,Z 438.108,A -85,B 0,C 180,E1 -25396.065,E2 -25396.065} C_VEL
LIN {X 0,Y 187.215,Z 442.025,A -85,B 0,C 180,E1 -25398.414,E2 -25398.414} C_VEL
LIN {X 0,Y 190.432,Z 447.858,A -85,B 0,C 180,E1 -25401.303,E2 -25401.303} C_VEL
LIN {X 0,Y 194.01,Z 454.91,A -85,B 0,C 180,E1 -25404.122,E2 -25404.122} C_VEL
LIN {X 0,Y 195.222,Z 457.541,A -85,B 0,C 180,E1 -25405.014,E2 -25405.014} C_VEL
LIN {X 0,Y 191.89,Z 492.653,A -85,B 0,C 180,E1 -25406.022,E2 -25406.022} C_VEL
LIN {X 0,Y 189.504,Z 506.445,A -85,B 0,C 180,E1 -25406.671,E2 -25406.671} C_VEL
LIN {X 0,Y 186.325,Z 519.437,A -85,B 0,C 180,E1 -25407.579,E2 -25407.579} C_VEL
LIN {X 0,Y 182.258,Z 531.836,A -85,B 0,C 180,E1 -25408.69,E2 -25408.69} C_VEL
LIN {X 0,Y 176.968,Z 544.804,A -85,B 0,C 180,E1 -25410.261,E2 -25410.261} C_VEL
LIN {X 0,Y 171.284,Z 556.32,A -85,B 0,C 180,E1 -25412.091,E2 -25412.091} C_VEL
LIN {X 0,Y 166.748,Z 564.305,A -85,B 0,C 180,E1 -25413.655,E2 -25413.655} C_VEL
LIN {X 0,Y 160.596,Z 573.725,A -85,B 0,C 180,E1 -25415.946,E2 -25415.946} C_VEL
LIN {X 0,Y 153.778,Z 583.173,A -85,B 0,C 180,E1 -25419.021,E2 -25419.021} C_VEL
LIN {X 0,Y 147.454,Z 590.987,A -85,B 0,C 180,E1 -25422.375,E2 -25422.375} C_VEL
LIN {X 0,Y 141.622,Z 597.451,A -85,B 0,C 180,E1 -25425.994,E2 -25425.994} C_VEL
LIN {X 0,Y 136.308,Z 602.785,A -85,B 0,C 180,E1 -25429.873,E2 -25429.873} C_VEL
LIN {X 0,Y 131.652,Z 607.139,A -85,B 0,C 180,E1 -25434.041,E2 -25434.041} C_VEL
LIN {X 0,Y 126.549,Z 611.503,A -85,B 0,C 180,E1 -25440.013,E2 -25440.013} C_VEL
LIN {X 0,Y 122.859,Z 614.392,A -85,B 0,C 180,E1 -25446.396,E2 -25446.396} C_VEL
LIN {X 0,Y 120.37,Z 615.903,A -85,B 0,C 180,E1 -25453.027,E2 -25453.027} C_VEL
LIN {X 0,Y 119.283,Z 616.073,A -85,B 0,C 180,E1 -25459.819,E2 -25459.819} C_VEL
LIN {X 0,Y 119.196,Z 615.661,A -85,B 0,C 180,E1 -25463.228,E2 -25463.228} C_VEL
LIN {X 0,Y 119.292,Z 614.923,A -85,B 0,C 180,E1 -25466.623,E2 -25466.623} C_VEL
LIN {X 0,Y 119.962,Z 612.457,A -85,B 0,C 180,E1 -25473.358,E2 -25473.358} C_VEL
LIN {X 0,Y 121.697,Z 608.594,A -85,B 0,C 180,E1 -25479.977,E2 -25479.977} C_VEL
LIN {X 0,Y 124.67,Z 603.18,A -85,B 0,C 180,E1 -25486.371,E2 -25486.371} C_VEL
LIN {X 0,Y 128.199,Z 597.598,A -85,B 0,C 180,E1 -25491.254,E2 -25491.254} C_VEL
LIN {X 0,Y 132.402,Z 590.641,A -85,B 0,C 180,E1 -25495.97,E2 -25495.97} C_VEL
LIN {X 0,Y 136.868,Z 582.935,A -85,B 0,C 180,E1 -25500.042,E2 -25500.042} C_VEL
LIN {X 0,Y 141.988,Z 573.649,A -85,B 0,C 180,E1 -25503.837,E2 -25503.837} C_VEL
LIN {X 0,Y 147.209,Z 563.367,A -85,B 0,C 180,E1 -25507.065,E2 -25507.065} C_VEL
LIN {X 0,Y 152.264,Z 552.039,A -85,B 0,C 180,E1 -25509.822,E2 -25509.822} C_VEL
LIN {X 0,Y 157.006,Z 539.513,A -85,B 0,C 180,E1 -25512.177,E2 -25512.177} C_VEL
LIN {X 0,Y 160.956,Z 527.352,A -85,B 0,C 180,E1 -25513.88,E2 -25513.88} C_VEL
LIN {X 0,Y 164.437,Z 513.932,A -85,B 0,C 180,E1 -25515.278,E2 -25515.278} C_VEL
LIN {X 0,Y 166.941,Z 500.485,A -85,B 0,C 180,E1 -25516.307,E2 -25516.307} C_VEL
LIN {X 0,Y 168.52,Z 487.633,A -85,B 0,C 180,E1 -25516.964,E2 -25516.964} C_VEL
LIN {X 0,Y 172.32,Z 438.452,A -85,B 0,C 180,E1 -25518.657,E2 -25518.657} C_VEL
LIN {X 0,Y 168.491,Z 430.323,A -85,B 0,C 180,E1 -25520.935,E2 -25520.935} C_VEL
LIN {X 0,Y 164.43,Z 422.82,A -85,B 0,C 180,E1 -25523.534,E2 -25523.534} C_VEL
LIN {X 0,Y 160.592,Z 416.334,A -85,B 0,C 180,E1 -25526.251,E2 -25526.251} C_VEL
LIN {X 0,Y 156.517,Z 409.913,A -85,B 0,C 180,E1 -25529.52,E2 -25529.52} C_VEL
LIN {X 0,Y 153.914,Z 406.081,A -85,B 0,C 180,E1 -25531.886,E2 -25531.886} C_VEL
LIN {X 0,Y 151.445,Z 402.439,A -85,B 0,C 180,E1 -25534.43,E2 -25534.43} C_VEL
LIN {X 0,Y 148.851,Z 398.893,A -85,B 0,C 180,E1 -25537.51,E2 -25537.51} C_VEL
LIN {X 0,Y 148.161,Z 397.929,A -85,B 0,C 180,E1 -25538.435,E2 -25538.435} C_VEL
LIN {X 0,Y 145.788,Z 395.283,A -85,B 0,C 180,E1 -25541.993,E2 -25541.993} C_VEL
LIN {X 0,Y 144.669,Z 392.991,A -85,B 0,C 180,E1 -25544.284,E2 -25544.284} C_VEL
LIN {X 0,Y 141.76,Z 389.841,A -85,B 0,C 180,E1 -25554.309,E2 -25554.309} C_VEL
LIN {X 0,Y 141.695,Z 389.282,A -85,B 0,C 180,E1 -25557.156,E2 -25557.156} C_VEL
LIN {X 0,Y 141.929,Z 389.647,A -85,B 0,C 180,E1 -25560.442,E2 -25560.442} C_VEL
LIN {X 0,Y 143.564,Z 392.122,A -85,B 0,C 180,E1 -25566.941,E2 -25566.941} C_VEL
LIN {X 0,Y 144.921,Z 393.206,A -85,B 0,C 180,E1 -25569.846,E2 -25569.846} C_VEL
LIN {X 0,Y 146.71,Z 396.425,A -85,B 0,C 180,E1 -25573.152,E2 -25573.152} C_VEL
LIN {X 0,Y 148.66,Z 398.519,A -85,B 0,C 180,E1 -25575.861,E2 -25575.861} C_VEL
LIN {X 0,Y 151.424,Z 402.433,A -85,B 0,C 180,E1 -25579.189,E2 -25579.189} C_VEL
LIN {X 0,Y 155.41,Z 408.146,A -85,B 0,C 180,E1 -25583.132,E2 -25583.132} C_VEL
LIN {X 0,Y 158.811,Z 413.333,A -85,B 0,C 180,E1 -25586,E2 -25586} C_VEL
LIN {X 0,Y 163.139,Z 420.579,A -85,B 0,C 180,E1 -25589.22,E2 -25589.22} C_VEL
LIN {X 0,Y 167.802,Z 431.422,A -85,B 0,C 180,E1 -25592.453,E2 -25592.453} C_VEL
LIN {X 0,Y 171.588,Z 441.941,A -85,B 0,C 180,E1 -25594.899,E2 -25594.899} C_VEL
LIN {X 0,Y 172.117,Z 443.856,A -85,B 0,C 180,E1 -25595.251,E2 -25595.251} C_VEL
LIN {X 0,Y 167.811,Z 496.614,A -85,B 0,C 180,E1 -25597.005,E2 -25597.005} C_VEL
LIN {X 0,Y 165.666,Z 511.114,A -85,B 0,C 180,E1 -25597.805,E2 -25597.805} C_VEL
LIN {X 0,Y 162.668,Z 524.879,A -85,B 0,C 180,E1 -25598.953,E2 -25598.953} C_VEL
LIN {X 0,Y 159.016,Z 537.312,A -85,B 0,C 180,E1 -25600.326,E2 -25600.326} C_VEL
LIN {X 0,Y 154.405,Z 550.331,A -85,B 0,C 180,E1 -25602.301,E2 -25602.301} C_VEL
LIN {X 0,Y 149.567,Z 562.154,A -85,B 0,C 180,E1 -25604.709,E2 -25604.709} C_VEL
LIN {X 0,Y 144.927,Z 571.969,A -85,B 0,C 180,E1 -25607.243,E2 -25607.243} C_VEL
LIN {X 0,Y 139.213,Z 582.821,A -85,B 0,C 180,E1 -25610.874,E2 -25610.874} C_VEL
LIN {X 0,Y 134.11,Z 591.775,A -85,B 0,C 180,E1 -25614.8,E2 -25614.8} C_VEL
LIN {X 0,Y 129.1,Z 600.354,A -85,B 0,C 180,E1 -25619.766,E2 -25619.766} C_VEL
LIN {X 0,Y 125.142,Z 607.264,A -85,B 0,C 180,E1 -25625.09,E2 -25625.09} C_VEL
LIN {X 0,Y 122.532,Z 612.014,A -85,B 0,C 180,E1 -25629.872,E2 -25629.872} C_VEL
LIN {X 0,Y 120.244,Z 616.927,A -85,B 0,C 180,E1 -25636.48,E2 -25636.48} C_VEL
LIN {X 0,Y 119.302,Z 620.327,A -85,B 0,C 180,E1 -25643.234,E2 -25643.234} C_VEL
LIN {X 0,Y 119.219,Z 621.49,A -85,B 0,C 180,E1 -25646.621,E2 -25646.621} C_VEL
LIN {X 0,Y 119.332,Z 622.302,A -85,B 0,C 180,E1 -25650,E2 -25650} C_VEL
LIN {X 0,Y 119.218,Z 622.759,A -85,B 0,C 180,E1 -25653.38,E2 -25653.38} C_VEL
LIN {X 0,Y 119.315,Z 622.864,A -85,B 0,C 180,E1 -25657.019,E2 -25657.019} C_VEL
LIN {X 0,Y 118.919,Z 622.692,A -85,B 0,C 180,E1 -25659.851,E2 -25659.851} C_VEL
LIN {X 0,Y 117.032,Z 621.896,A -85,B 0,C 180,E1 -25664.567,E2 -25664.567} C_VEL
LIN {X 0,Y 115.915,Z 620.922,A -85,B 0,C 180,E1 -25668.414,E2 -25668.414} C_VEL
LIN {X 0,Y 116.177,Z 619.917,A -85,B 0,C 180,E1 -25671.292,E2 -25671.292} C_VEL
LIN {X 0,Y 116.585,Z 619.5,A -85,B 0,C 180,E1 -25672.222,E2 -25672.222} C_VEL
LIN {X 0,Y 120.326,Z 616.504,A -85,B 0,C 180,E1 -25677.856,E2 -25677.856} C_VEL
LIN {X 0,Y 124.333,Z 613,A -85,B 0,C 180,E1 -25682.478,E2 -25682.478} C_VEL
LIN {X 0,Y 130.989,Z 606.932,A -85,B 0,C 180,E1 -25688.097,E2 -25688.097} C_VEL
LIN {X 0,Y 137.759,Z 600.146,A -85,B 0,C 180,E1 -25692.528,E2 -25692.528} C_VEL
LIN {X 0,Y 145.386,Z 591.736,A -85,B 0,C 180,E1 -25696.476,E2 -25696.476} C_VEL
LIN {X 0,Y 153.123,Z 581.943,A -85,B 0,C 180,E1 -25699.878,E2 -25699.878} C_VEL
LIN {X 0,Y 159.688,Z 572.412,A -85,B 0,C 180,E1 -25702.389,E2 -25702.389} C_VEL
LIN {X 0,Y 166.18,Z 561.75,A -85,B 0,C 180,E1 -25704.497,E2 -25704.497} C_VEL
LIN {X 0,Y 172.199,Z 550.129,A -85,B 0,C 180,E1 -25706.258,E2 -25706.258} C_VEL
LIN {X 0,Y 177.769,Z 537.342,A -85,B 0,C 180,E1 -25707.675,E2 -25707.675} C_VEL
LIN {X 0,Y 182.297,Z 524.156,A -85,B 0,C 180,E1 -25708.781,E2 -25708.781} C_VEL
LIN {X 0,Y 185.939,Z 510.142,A -85,B 0,C 180,E1 -25709.618,E2 -25709.618} C_VEL
LIN {X 0,Y 188.438,Z 495.689,A -85,B 0,C 180,E1 -25710.193,E2 -25710.193} C_VEL
LIN {X 0,Y 191.342,Z 465.302,A -85,B 0,C 180,E1 -25711.047,E2 -25711.047} C_VEL
LIN {X 0,Y 188.457,Z 457.207,A -85,B 0,C 180,E1 -25713.62,E2 -25713.62} C_VEL
LIN {X 0,Y 185.374,Z 449.266,A -85,B 0,C 180,E1 -25716.736,E2 -25716.736} C_VEL
LIN {X 0,Y 182.772,Z 443.503,A -85,B 0,C 180,E1 -25719.754,E2 -25719.754} C_VEL
LIN {X 0,Y 180.23,Z 439.309,A -85,B 0,C 180,E1 -25723.179,E2 -25723.179} C_VEL
LIN {X 0,Y 178.179,Z 435.612,A -85,B 0,C 180,E1 -25726.892,E2 -25726.892} C_VEL
LIN {X 0,Y 176.356,Z 432.52,A -85,B 0,C 180,E1 -25732.132,E2 -25732.132} C_VEL
LIN {X 0,Y 176.1,Z 431.186,A -85,B 0,C 180,E1 -25734,E2 -25734} C_VEL
LIN {X 0,Y 176.157,Z 430.994,A -85,B 0,C 180,E1 -25740.624,E2 -25740.624} C_VEL
LIN {X 0,Y 177.686,Z 434.885,A -85,B 0,C 180,E1 -25746.459,E2 -25746.459} C_VEL
LIN {X 0,Y 178.406,Z 435.904,A -85,B 0,C 180,E1 -25747.997,E2 -25747.997} C_VEL
LIN {X 0,Y 180.89,Z 440.413,A -85,B 0,C 180,E1 -25752.233,E2 -25752.233} C_VEL
LIN {X 0,Y 183.347,Z 444.683,A -85,B 0,C 180,E1 -25755.387,E2 -25755.387} C_VEL
LIN {X 0,Y 186.29,Z 449.949,A -85,B 0,C 180,E1 -25758.508,E2 -25758.508} C_VEL
LIN {X 0,Y 190.437,Z 458.267,A -85,B 0,C 180,E1 -25762.228,E2 -25762.228} C_VEL
LIN {X 0,Y 191.652,Z 460.917,A -85,B 0,C 180,E1 -25763.213,E2 -25763.213} C_VEL
LIN {X 0,Y 188.544,Z 492.85,A -85,B 0,C 180,E1 -25764.143,E2 -25764.143} C_VEL
LIN {X 0,Y 186.243,Z 505.965,A -85,B 0,C 180,E1 -25764.74,E2 -25764.74} C_VEL
LIN {X 0,Y 183.111,Z 518.634,A -85,B 0,C 180,E1 -25765.587,E2 -25765.587} C_VEL
LIN {X 0,Y 178.924,Z 531.253,A -85,B 0,C 180,E1 -25766.674,E2 -25766.674} C_VEL
LIN {X 0,Y 174.162,Z 542.938,A -85,B 0,C 180,E1 -25768.03,E2 -25768.03} C_VEL
LIN {X 0,Y 168.706,Z 553.9,A -85,B 0,C 180,E1 -25769.617,E2 -25769.617} C_VEL
LIN {X 0,Y 162.227,Z 565.068,A -85,B 0,C 180,E1 -25771.77,E2 -25771.77} C_VEL
LIN {X 0,Y 155.251,Z 575.249,A -85,B 0,C 180,E1 -25774.297,E2 -25774.297} C_VEL
LIN {X 0,Y 148.19,Z 584.447,A -85,B 0,C 180,E1 -25777.406,E2 -25777.406} C_VEL
LIN {X 0,Y 141.542,Z 592.161,A -85,B 0,C 180,E1 -25780.857,E2 -25780.857} C_VEL
LIN {X 0,Y 134.575,Z 599.343,A -85,B 0,C 180,E1 -25785.171,E2 -25785.171} C_VEL
LIN {X 0,Y 127.769,Z 605.555,A -85,B 0,C 180,E1 -25790.363,E2 -25790.363} C_VEL
LIN {X 0,Y 122.956,Z 609.597,A -85,B 0,C 180,E1 -25795.14,E2 -25795.14} C_VEL
LIN {X 0,Y 118.097,Z 613.249,A -85,B 0,C 180,E1 -25801.571,E2 -25801.571} C_VEL
LIN {X 0,Y 114.696,Z 615.476,A -85,B 0,C 180,E1 -25808.43,E2 -25808.43} C_VEL
LIN {X 0,Y 112.656,Z 616.35,A -85,B 0,C 180,E1 -25815.55,E2 -25815.55} C_VEL
LIN {X 0,Y 112.101,Z 615.891,A -85,B 0,C 180,E1 -25822.797,E2 -25822.797} C_VEL
LIN {X 0,Y 112.171,Z 615.17,A -85,B 0,C 180,E1 -25826.408,E2 -25826.408} C_VEL
LIN {X 0,Y 112.454,Z 613.995,A -85,B 0,C 180,E1 -25830.403,E2 -25830.403} C_VEL
LIN {X 0,Y 113.609,Z 611.014,A -85,B 0,C 180,E1 -25837.107,E2 -25837.107} C_VEL
LIN {X 0,Y 116.16,Z 606.446,A -85,B 0,C 180,E1 -25844.005,E2 -25844.005} C_VEL
LIN {X 0,Y 118.981,Z 601.954,A -85,B 0,C 180,E1 -25848.957,E2 -25848.957} C_VEL
LIN {X 0,Y 123.274,Z 595.473,A -85,B 0,C 180,E1 -25854.414,E2 -25854.414} C_VEL
LIN {X 0,Y 128.299,Z 587.455,A -85,B 0,C 180,E1 -25859.537,E2 -25859.537} C_VEL
LIN {X 0,Y 133.45,Z 579.047,A -85,B 0,C 180,E1 -25863.57,E2 -25863.57} C_VEL
LIN {X 0,Y 139.121,Z 568.901,A -85,B 0,C 180,E1 -25867.314,E2 -25867.314} C_VEL
LIN {X 0,Y 144.807,Z 557.536,A -85,B 0,C 180,E1 -25870.475,E2 -25870.475} C_VEL
LIN {X 0,Y 149.641,Z 546.242,A -85,B 0,C 180,E1 -25872.921,E2 -25872.921} C_VEL
LIN {X 0,Y 154.17,Z 533.884,A -85,B 0,C 180,E1 -25874.956,E2 -25874.956} C_VEL
LIN {X 0,Y 158.352,Z 520.067,A -85,B 0,C 180,E1 -25876.613,E2 -25876.613} C_VEL
LIN {X 0,Y 161.501,Z 506.061,A -85,B 0,C 180,E1 -25877.844,E2 -25877.844} C_VEL
LIN {X 0,Y 163.656,Z 491.686,A -85,B 0,C 180,E1 -25878.716,E2 -25878.716} C_VEL
LIN {X 0,Y 167.769,Z 440.976,A -85,B 0,C 180,E1 -25880.513,E2 -25880.513} C_VEL
LIN {X 0,Y 163.253,Z 431.61,A -85,B 0,C 180,E1 -25883.473,E2 -25883.473} C_VEL
LIN {X 0,Y 158.739,Z 423.369,A -85,B 0,C 180,E1 -25886.777,E2 -25886.777} C_VEL
LIN {X 0,Y 154.257,Z 416.028,A -85,B 0,C 180,E1 -25890.561,E2 -25890.561} C_VEL
LIN {X 0,Y 151.731,Z 412.174,A -85,B 0,C 180,E1 -25893.018,E2 -25893.018} C_VEL
LIN {X 0,Y 149.517,Z 408.804,A -85,B 0,C 180,E1 -25895.464,E2 -25895.464} C_VEL
LIN {X 0,Y 146.661,Z 404.645,A -85,B 0,C 180,E1 -25899.193,E2 -25899.193} C_VEL
LIN {X 0,Y 144.399,Z 401.911,A -85,B 0,C 180,E1 -25902.837,E2 -25902.837} C_VEL
LIN {X 0,Y 143.476,Z 399.91,A -85,B 0,C 180,E1 -25904.878,E2 -25904.878} C_VEL
LIN {X 0,Y 140.894,Z 396.906,A -85,B 0,C 180,E1 -25914.273,E2 -25914.273} C_VEL
LIN {X 0,Y 140.825,Z 396.362,A -85,B 0,C 180,E1 -25917.138,E2 -25917.138} C_VEL
LIN {X 0,Y 141.047,Z 396.805,A -85,B 0,C 180,E1 -25920.445,E2 -25920.445} C_VEL
LIN {X 0,Y 142.7,Z 399.187,A -85,B 0,C 180,E1 -25926.983,E2 -25926.983} C_VEL
LIN {X 0,Y 143.668,Z 400.025,A -85,B 0,C 180,E1 -25929.148,E2 -25929.148} C_VEL
LIN {X 0,Y 145.358,Z 403.154,A -85,B 0,C 180,E1 -25932.477,E2 -25932.477} C_VEL
LIN {X 0,Y 147.083,Z 405.17,A -85,B 0,C 180,E1 -25935.036,E2 -25935.036} C_VEL
LIN {X 0,Y 149.78,Z 409.059,A -85,B 0,C 180,E1 -25938.464,E2 -25938.464} C_VEL
LIN {X 0,Y 153.336,Z 414.524,A -85,B 0,C 180,E1 -25942.206,E2 -25942.206} C_VEL
LIN {X 0,Y 156.987,Z 420.254,A -85,B 0,C 180,E1 -25945.437,E2 -25945.437} C_VEL
LIN {X 0,Y 160.588,Z 426.878,A -85,B 0,C 180,E1 -25948.284,E2 -25948.284} C_VEL
LIN {X 0,Y 164.869,Z 437.667,A -85,B 0,C 180,E1 -25951.471,E2 -25951.471} C_VEL
LIN {X 0,Y 167.576,Z 445.608,A -85,B 0,C 180,E1 -25953.362,E2 -25953.362} C_VEL
LIN {X 0,Y 163.25,Z 497.236,A -85,B 0,C 180,E1 -25955.121,E2 -25955.121} C_VEL
LIN {X 0,Y 160.926,Z 512.008,A -85,B 0,C 180,E1 -25955.975,E2 -25955.975} C_VEL
LIN {X 0,Y 157.64,Z 526.053,A -85,B 0,C 180,E1 -25957.166,E2 -25957.166} C_VEL
LIN {X 0,Y 153.884,Z 538.189,A -85,B 0,C 180,E1 -25958.548,E2 -25958.548} C_VEL
LIN {X 0,Y 149.095,Z 551,A -85,B 0,C 180,E1 -25960.529,E2 -25960.529} C_VEL
LIN {X 0,Y 144.063,Z 562.669,A -85,B 0,C 180,E1 -25962.968,E2 -25962.968} C_VEL
LIN {X 0,Y 138.701,Z 573.346,A -85,B 0,C 180,E1 -25965.838,E2 -25965.838} C_VEL
LIN {X 0,Y 132.778,Z 583.938,A -85,B 0,C 180,E1 -25969.581,E2 -25969.581} C_VEL
LIN {X 0,Y 127.488,Z 592.672,A -85,B 0,C 180,E1 -25973.659,E2 -25973.659} C_VEL
LIN {X 0,Y 122.282,Z 601.044,A -85,B 0,C 180,E1 -25978.852,E2 -25978.852} C_VEL
LIN {X 0,Y 118.672,Z 606.881,A -85,B 0,C 180,E1 -25983.631,E2 -25983.631} C_VEL
LIN {X 0,Y 115.838,Z 611.67,A -85,B 0,C 180,E1 -25988.653,E2 -25988.653} C_VEL
LIN {X 0,Y 113.304,Z 616.619,A -85,B 0,C 180,E1 -25995.635,E2 -25995.635} C_VEL
LIN {X 0,Y 112.234,Z 620.054,A -85,B 0,C 180,E1 -26002.806,E2 -26002.806} C_VEL
LIN {X 0,Y 112.124,Z 621.234,A -85,B 0,C 180,E1 -26006.406,E2 -26006.406} C_VEL
LIN {X 0,Y 112.248,Z 622.067,A -85,B 0,C 180,E1 -26010,E2 -26010} C_VEL
LIN {X 0,Y 112.237,Z 622.681,A -85,B 0,C 180,E1 -26017.194,E2 -26017.194} C_VEL
LIN {X 0,Y 113.405,Z 621.964,A -85,B 0,C 180,E1 -26024.352,E2 -26024.352} C_VEL
LIN {X 0,Y 116.096,Z 619.92,A -85,B 0,C 180,E1 -26031.297,E2 -26031.297} C_VEL
LIN {X 0,Y 116.585,Z 619.5,A -85,B 0,C 180,E1 -26032.222,E2 -26032.222} C_VEL
LIN {X 0,Y 117.546,Z 618.258,A -85,B 0,C 180,E1 -26035.004,E2 -26035.004} C_VEL
LIN {X 0,Y 117.925,Z 615.789,A -85,B 0,C 180,E1 -26039.683,E2 -26039.683} C_VEL
LIN {X 0,Y 118.622,Z 613.483,A -85,B 0,C 180,E1 -26043.354,E2 -26043.354} C_VEL
LIN {X 0,Y 120.194,Z 611.474,A -85,B 0,C 180,E1 -26045.913,E2 -26045.913} C_VEL
LIN {X 0,Y 121.014,Z 610.729,A -85,B 0,C 180,E1 -26046.692,E2 -26046.692} C_VEL
LIN {X 0,Y 127.416,Z 605.097,A -85,B 0,C 180,E1 -26051.443,E2 -26051.443} C_VEL
LIN {X 0,Y 134.792,Z 597.933,A -85,B 0,C 180,E1 -26055.799,E2 -26055.799} C_VEL
LIN {X 0,Y 142.973,Z 589.097,A -85,B 0,C 180,E1 -26059.632,E2 -26059.632} C_VEL
LIN {X 0,Y 150.324,Z 579.863,A -85,B 0,C 180,E1 -26062.633,E2 -26062.633} C_VEL
LIN {X 0,Y 157.46,Z 569.672,A -85,B 0,C 180,E1 -26065.097,E2 -26065.097} C_VEL
LIN {X 0,Y 164.187,Z 558.474,A -85,B 0,C 180,E1 -26067.142,E2 -26067.142} C_VEL
LIN {X 0,Y 170.507,Z 546.103,A -85,B 0,C 180,E1 -26068.788,E2 -26068.788} C_VEL
LIN {X 0,Y 175.513,Z 534.203,A -85,B 0,C 180,E1 -26069.985,E2 -26069.985} C_VEL
LIN {X 0,Y 180.135,Z 520.195,A -85,B 0,C 180,E1 -26071.027,E2 -26071.027} C_VEL
LIN {X 0,Y 183.652,Z 505.488,A -85,B 0,C 180,E1 -26071.796,E2 -26071.796} C_VEL
LIN {X 0,Y 185.774,Z 491.685,A -85,B 0,C 180,E1 -26072.259,E2 -26072.259} C_VEL
LIN {X 0,Y 187.952,Z 468.227,A -85,B 0,C 180,E1 -26072.953,E2 -26072.953} C_VEL
LIN {X 0,Y 185.331,Z 460.499,A -85,B 0,C 180,E1 -26075.588,E2 -26075.588} C_VEL
LIN {X 0,Y 182.905,Z 454.124,A -85,B 0,C 180,E1 -26078.322,E2 -26078.322} C_VEL
LIN {X 0,Y 181.096,Z 449.87,A -85,B 0,C 180,E1 -26080.629,E2 -26080.629} C_VEL
LIN {X 0,Y 178.859,Z 445.96,A -85,B 0,C 180,E1 -26083.871,E2 -26083.871} C_VEL
LIN {X 0,Y 177.01,Z 442.468,A -85,B 0,C 180,E1 -26087.46,E2 -26087.46} C_VEL
LIN {X 0,Y 175.311,Z 439.056,A -85,B 0,C 180,E1 -26093.093,E2 -26093.093} C_VEL
LIN {X 0,Y 175.134,Z 438.172,A -85,B 0,C 180,E1 -26094.683,E2 -26094.683} C_VEL
LIN {X 0,Y 175.253,Z 438.041,A -85,B 0,C 180,E1 -26100.418,E2 -26100.418} C_VEL
LIN {X 0,Y 176.491,Z 441.596,A -85,B 0,C 180,E1 -26105.715,E2 -26105.715} C_VEL
LIN {X 0,Y 177.22,Z 442.668,A -85,B 0,C 180,E1 -26107.406,E2 -26107.406} C_VEL
LIN {X 0,Y 179.411,Z 446.912,A -85,B 0,C 180,E1 -26111.439,E2 -26111.439} C_VEL
LIN {X 0,Y 181.731,Z 451.176,A -85,B 0,C 180,E1 -26114.631,E2 -26114.631} C_VEL
LIN {X 0,Y 184.333,Z 456.1,A -85,B 0,C 180,E1 -26117.581,E2 -26117.581} C_VEL
LIN {X 0,Y 188.12,Z 464.086,A -85,B 0,C 180,E1 -26121.22,E2 -26121.22} C_VEL
LIN {X 0,Y 188.302,Z 464.467,A -85,B 0,C 180,E1 -26121.377,E2 -26121.377} C_VEL
LIN {X 0,Y 185.352,Z 493.341,A -85,B 0,C 180,E1 -26122.202,E2 -26122.202} C_VEL
LIN {X 0,Y 182.956,Z 506.499,A -85,B 0,C 180,E1 -26122.794,E2 -26122.794} C_VEL
LIN {X 0,Y 179.415,Z 520.116,A -85,B 0,C 180,E1 -26123.707,E2 -26123.707} C_VEL
LIN {X 0,Y 174.407,Z 534.239,A -85,B 0,C 180,E1 -26124.954,E2 -26124.954} C_VEL
LIN {X 0,Y 168.779,Z 546.817,A -85,B 0,C 180,E1 -26126.461,E2 -26126.461} C_VEL
